// TIA Portal V20 export
FUNCTION_BLOCK "Sequence_2_TopTapeAttachment"   // FB32849, LAD
TITLE = Sequence
// Sequence template programmend in ladder logic
// stored: IsIECCheckEnabled true, MemoryReserve 100, Namespace Unit1.Em3, SetENOAutomatically true
   VAR_INPUT
      unitStatus : "LAF_typeUnitStatus";
   END_VAR
   VAR
      instSequenceLADControl { ExternalWritable := 'False'} : "LAF_ControlLadSequence";
      instSequenceLADStatus { ExternalWritable := 'False'} : "LAF_StatusLadSequence";
      statTonTime { ExternalWritable := 'False'} : Array[0..9999] of TON_TIME;
   END_VAR
   VAR_TEMP
      tempCustomerAction : Bool;   // Placeholder for possible actions
      tempDo_nothing_and_wait_for_init : Bool;   // Placeholder for doing nothing
      tempSafeStateCondition : Bool;   // Temp Condition for the equipment module to be in a safe state
   END_VAR
   VAR CONSTANT
      delayTime : Time := T#100ms;
      STEP_IDLE : DInt := 1;
      JOB_1_STEP_00 : DInt := 100;
      JOB_1_STEP_01 : DInt := 101;
      JOB_1_STEP_10 : DInt := 110;
      JOB_1_STEP_20 : DInt := 120;
      JOB_1_STEP_30 : DInt := 130;
      JOB_1_STEP_40 : DInt := 140;
      JOB_1_STEP_50 : DInt := 150;
      JOB_1_STEP_60 : DInt := 160;
      JOB_1_STEP_70 : DInt := 170;
      JOB_1_STEP_80 : DInt := 180;
      JOB_1_STEP_90 : DInt := 190;
      JOB_2_STEP_00 : DInt := 200;
      JOB_2_STEP_01 : DInt := 201;
      JOB_2_STEP_10 : DInt := 210;
      JOB_2_STEP_20 : DInt := 220;
      JOB_2_STEP_30 : DInt := 230;
      JOB_2_STEP_40 : DInt := 240;
      JOB_2_STEP_41 : DInt := 241;
      JOB_2_STEP_42 : DInt := 242;
      JOB_2_STEP_50 : DInt := 250;
      JOB_2_STEP_60 : DInt := 260;
      JOB_2_STEP_70 : DInt := 270;
      JOB_2_STEP_80 : DInt := 280;
      JOB_2_STEP_90 : DInt := 290;
      JOB_3_STEP_00 : DInt := 300;
      JOB_3_STEP_01 : DInt := 301;
      JOB_3_STEP_10 : DInt := 310;
      JOB_3_STEP_20 : DInt := 320;
      JOB_3_STEP_30 : DInt := 330;
      JOB_3_STEP_40 : DInt := 340;
      JOB_3_STEP_50 : DInt := 350;
      JOB_3_STEP_60 : DInt := 360;
      JOB_3_STEP_70 : DInt := 370;
      JOB_3_STEP_80 : DInt := 380;
      JOB_3_STEP_90 : DInt := 390;
      JOB_4_STEP_00 : DInt := 400;
      JOB_4_STEP_01 : DInt := 401;
      JOB_4_STEP_10 : DInt := 410;
      JOB_4_STEP_20 : DInt := 420;
      JOB_4_STEP_30 : DInt := 430;
      JOB_4_STEP_40 : DInt := 440;
      JOB_4_STEP_50 : DInt := 450;
      JOB_4_STEP_60 : DInt := 460;
      JOB_4_STEP_70 : DInt := 470;
      JOB_4_STEP_80 : DInt := 480;
      JOB_4_STEP_90 : DInt := 490;
      JOB_5_STEP_01 : DInt := 501;
      JOB_5_STEP_10 : DInt := 510;
      JOB_5_STEP_20 : DInt := 520;
      JOB_5_STEP_30 : DInt := 530;
      JOB_5_STEP_40 : DInt := 540;
      JOB_5_STEP_50 : DInt := 550;
      JOB_5_STEP_60 : DInt := 560;
      JOB_5_STEP_70 : DInt := 570;
      JOB_5_STEP_80 : DInt := 580;
      JOB_5_STEP_90 : DInt := 590;
      JOB_12_STEP_10 : DInt := 1210;
      JOB_12_STEP_20 : DInt := 1220;
      JOB_12_STEP_30 : DInt := 1230;
      JOB_12_STEP_40 : DInt := 1240;
      JOB_12_STEP_50 : DInt := 1250;
      JOB_12_STEP_60 : DInt := 1260;
      JOB_12_STEP_70 : DInt := 1270;
      JOB_12_STEP_80 : DInt := 1280;
      JOB_12_STEP_90 : DInt := 1290;
      JOB_13_STEP_00 : DInt := 1300;
      JOB_13_STEP_10 : DInt := 1310;
      JOB_13_STEP_20 : DInt := 1320;
      JOB_13_STEP_30 : DInt := 1330;
      JOB_13_STEP_40 : DInt := 1340;
      JOB_13_STEP_50 : DInt := 1350;
      JOB_13_STEP_60 : DInt := 1360;
      JOB_13_STEP_70 : DInt := 1370;
      JOB_13_STEP_80 : DInt := 1380;
      JOB_13_STEP_90 : DInt := 1390;
      STEP_IMMEDIATE_STOP : DInt := 9001;   // Step executed when an immediate stop command is triggered for the sequence (i.e. when unit is in state aborting)
      TO_DO_INSERT_ACTIONS_HERE : Bool := TRUE;   // Template : Add actions
      TO_DO_INSERT_CONDITION_FOR_TRANSITION_HERE : Bool := TRUE;   // Template : Add conditions
   END_VAR
   VAR_TEMP   // added for the SCL form of the ladder/FBD networks
      _w1 : Bool;
   END_VAR
BEGIN

REGION Network 1: BLOCK INFO HEADER
   // (company) / (C) Copyright (year)
   // ---------------------------------------------------------------------------------
   // Title:                             (Title of this block)
   // Comment/Function: (that is implemented in the block)
   // Library/Family:           (that the source is dedicated to)
   // Author:                        (department / person in charge / contact)
   // Target System:          (test system with FW version)
   // Engineering:              TIA Portal (SW version)
   // Restrictions:               (OB types, etc.)
   // Requirements:           (hardware, technological package, etc.)
   // ---------------------------------------------------------------------------------
   // Change log table:
   // Version          | Date             | Signature      | Expert in charge  | Changes applied ------------------------|----------------------|-------------------------|--------------------------------|-----------------------
   // 001.000.000 | yyyy-mm-dd | 0x00000000 | (name of expert) | First released version
END_REGION

REGION Network 2: DESCRIPTION
   // This is a template block provided by the Automation Framework. It can be used to create an own project.
   // The Block Info Header is prepared to put in your own data.
   // Description of the block could be added here and the docu created by Code2Docu.
END_REGION

REGION Network 3: *************** CONTROL **********************
END_REGION

REGION Network 4: Sequence Control ("Enter your Sequins number here")
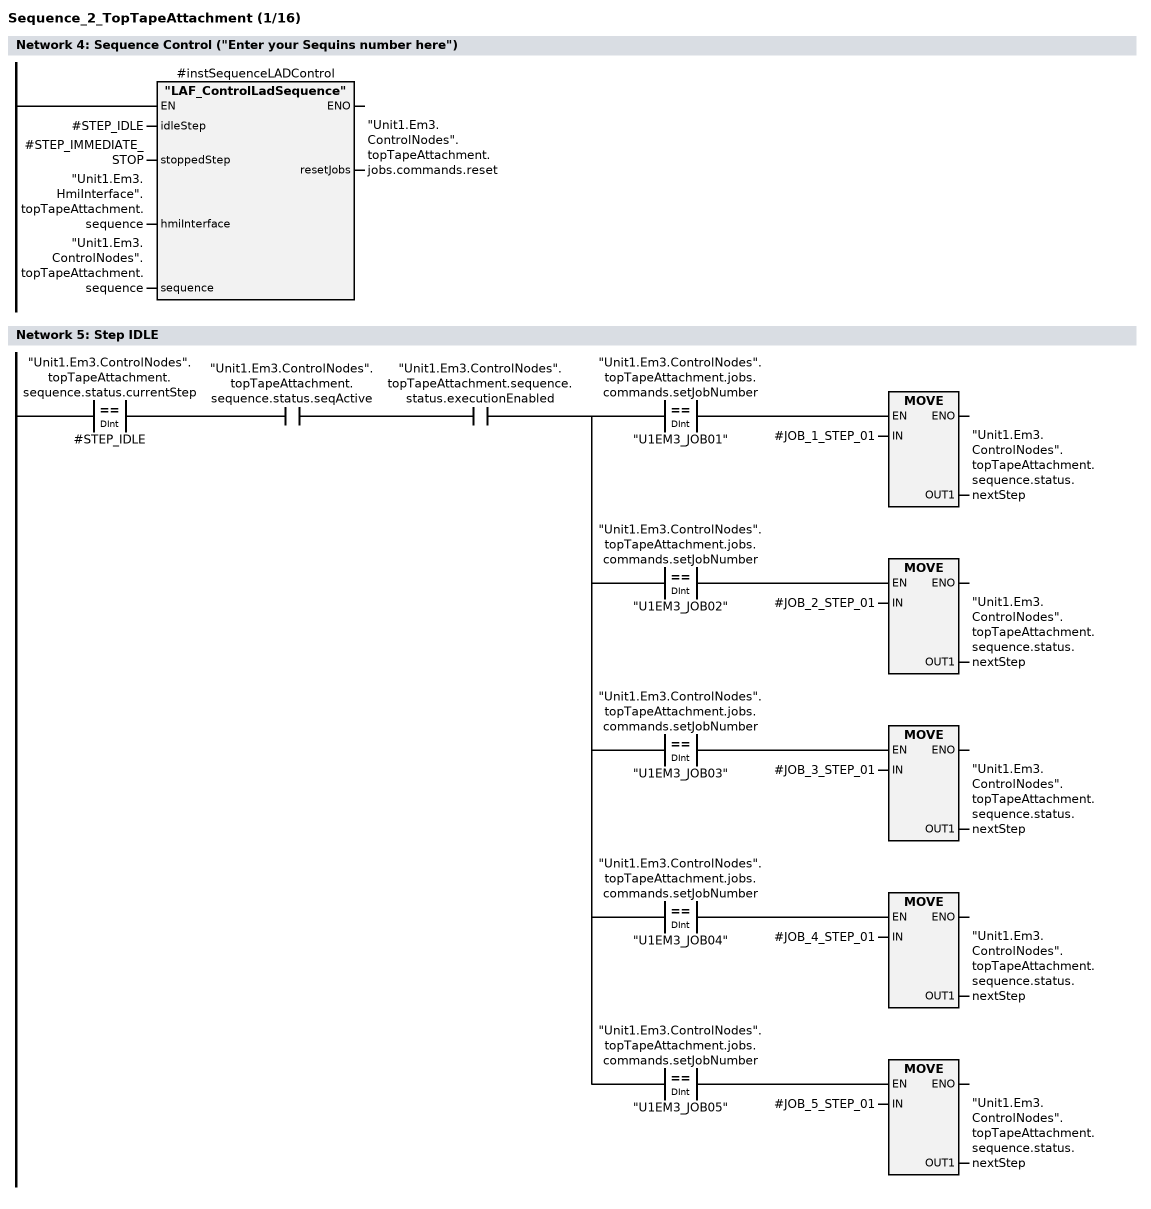
   RUNG wire#powerrail
      #instSequenceLADControl(idleStep := #STEP_IDLE, stoppedStep := #STEP_IMMEDIATE_STOP, hmiInterface := "Unit1.Em3.HmiInterface".topTapeAttachment.sequence, sequence := "Unit1.Em3.ControlNodes".topTapeAttachment.sequence, resetJobs => "Unit1.Em3.ControlNodes".topTapeAttachment.jobs.commands.reset)
   END_RUNG
   // the same network as SCL:
   #instSequenceLADControl(idleStep := #STEP_IDLE,   // "LAF_ControlLadSequence"
                           stoppedStep := #STEP_IMMEDIATE_STOP,
                           hmiInterface := "Unit1.Em3.HmiInterface".topTapeAttachment.sequence,
                           sequence := "Unit1.Em3.ControlNodes".topTapeAttachment.sequence,
                           resetJobs => "Unit1.Em3.ControlNodes".topTapeAttachment.jobs.commands.reset);
END_REGION

REGION Network 5: Step IDLE
   RUNG wire#powerrail
      { S7_Templates := "SrcType := DInt" } EQ_Contact(in1 := "Unit1.Em3.ControlNodes".topTapeAttachment.sequence.status.currentStep, in2 := #STEP_IDLE)
      Contact( "Unit1.Em3.ControlNodes".topTapeAttachment.sequence.status.seqActive )
      Contact( "Unit1.Em3.ControlNodes".topTapeAttachment.sequence.status.executionEnabled )
      wire#w1
      { S7_Templates := "SrcType := DInt" } EQ_Contact(in1 := "Unit1.Em3.ControlNodes".topTapeAttachment.jobs.commands.setJobNumber, in2 := "U1EM3_JOB01")
      Move(in := #JOB_1_STEP_01, out1 => "Unit1.Em3.ControlNodes".topTapeAttachment.sequence.status.nextStep)
   END_RUNG
   RUNG wire#w1
      { S7_Templates := "SrcType := DInt" } EQ_Contact(in1 := "Unit1.Em3.ControlNodes".topTapeAttachment.jobs.commands.setJobNumber, in2 := "U1EM3_JOB02")
      Move(in := #JOB_2_STEP_01, out1 => "Unit1.Em3.ControlNodes".topTapeAttachment.sequence.status.nextStep)
   END_RUNG
   RUNG wire#w1
      { S7_Templates := "SrcType := DInt" } EQ_Contact(in1 := "Unit1.Em3.ControlNodes".topTapeAttachment.jobs.commands.setJobNumber, in2 := "U1EM3_JOB03")
      Move(in := #JOB_3_STEP_01, out1 => "Unit1.Em3.ControlNodes".topTapeAttachment.sequence.status.nextStep)
   END_RUNG
   RUNG wire#w1
      { S7_Templates := "SrcType := DInt" } EQ_Contact(in1 := "Unit1.Em3.ControlNodes".topTapeAttachment.jobs.commands.setJobNumber, in2 := "U1EM3_JOB04")
      Move(in := #JOB_4_STEP_01, out1 => "Unit1.Em3.ControlNodes".topTapeAttachment.sequence.status.nextStep)
   END_RUNG
   RUNG wire#w1
      { S7_Templates := "SrcType := DInt" } EQ_Contact(in1 := "Unit1.Em3.ControlNodes".topTapeAttachment.jobs.commands.setJobNumber, in2 := "U1EM3_JOB05")
      Move(in := #JOB_5_STEP_01, out1 => "Unit1.Em3.ControlNodes".topTapeAttachment.sequence.status.nextStep)
   END_RUNG
   // the same network as SCL:
   #_w1 := ("Unit1.Em3.ControlNodes".topTapeAttachment.sequence.status.currentStep = #STEP_IDLE) AND "Unit1.Em3.ControlNodes".topTapeAttachment.sequence.status.seqActive AND "Unit1.Em3.ControlNodes".topTapeAttachment.sequence.status.executionEnabled;
   IF #_w1 AND ("Unit1.Em3.ControlNodes".topTapeAttachment.jobs.commands.setJobNumber = "U1EM3_JOB01") THEN
       "Unit1.Em3.ControlNodes".topTapeAttachment.sequence.status.nextStep := #JOB_1_STEP_01;
   END_IF;
   IF #_w1 AND ("Unit1.Em3.ControlNodes".topTapeAttachment.jobs.commands.setJobNumber = "U1EM3_JOB02") THEN
       "Unit1.Em3.ControlNodes".topTapeAttachment.sequence.status.nextStep := #JOB_2_STEP_01;
   END_IF;
   IF #_w1 AND ("Unit1.Em3.ControlNodes".topTapeAttachment.jobs.commands.setJobNumber = "U1EM3_JOB03") THEN
       "Unit1.Em3.ControlNodes".topTapeAttachment.sequence.status.nextStep := #JOB_3_STEP_01;
   END_IF;
   IF #_w1 AND ("Unit1.Em3.ControlNodes".topTapeAttachment.jobs.commands.setJobNumber = "U1EM3_JOB04") THEN
       "Unit1.Em3.ControlNodes".topTapeAttachment.sequence.status.nextStep := #JOB_4_STEP_01;
   END_IF;
   IF #_w1 AND ("Unit1.Em3.ControlNodes".topTapeAttachment.jobs.commands.setJobNumber = "U1EM3_JOB05") THEN
       "Unit1.Em3.ControlNodes".topTapeAttachment.sequence.status.nextStep := #JOB_5_STEP_01;
   END_IF;
END_REGION

REGION Network 6: *************** JOB[1] EM HOMING *************************
END_REGION

REGION Network 7: Step[101] : JOB[1] Condition
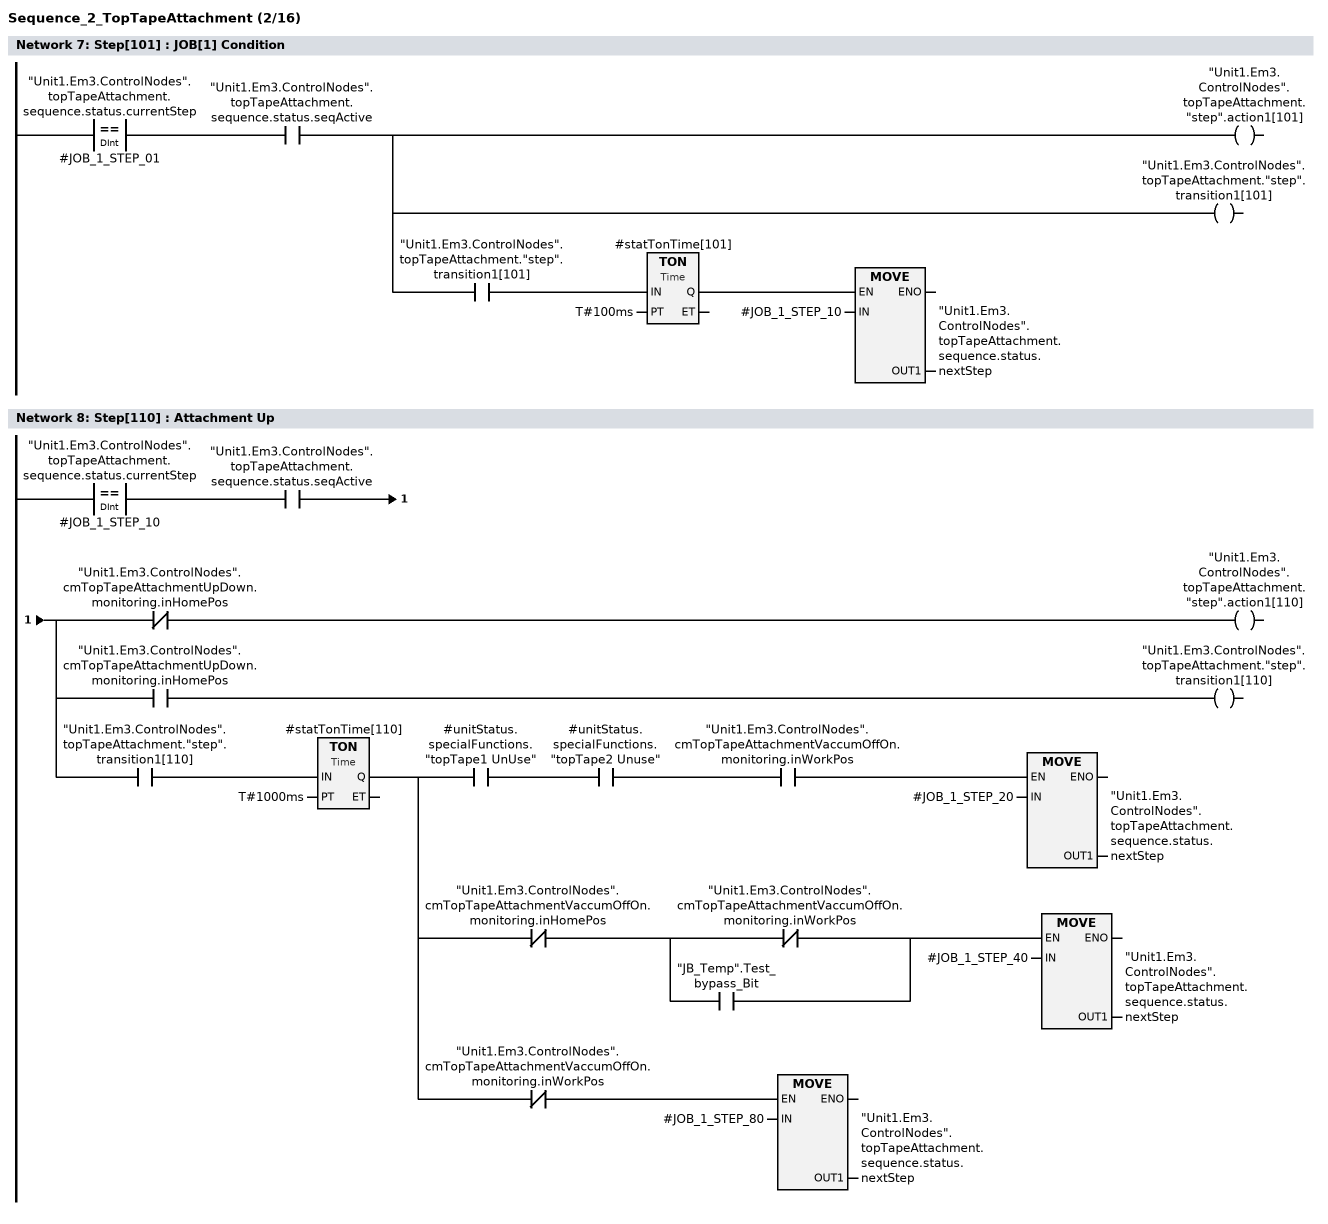
   RUNG wire#powerrail
      { S7_Templates := "SrcType := DInt" } EQ_Contact(in1 := "Unit1.Em3.ControlNodes".topTapeAttachment.sequence.status.currentStep, in2 := #JOB_1_STEP_01)
      Contact( "Unit1.Em3.ControlNodes".topTapeAttachment.sequence.status.seqActive )
      wire#w1
      Coil( "Unit1.Em3.ControlNodes".topTapeAttachment."step".action1[101] )
   END_RUNG
   RUNG wire#w1
      Coil( "Unit1.Em3.ControlNodes".topTapeAttachment."step".transition1[101] )
   END_RUNG
   RUNG wire#w1
      Contact( "Unit1.Em3.ControlNodes".topTapeAttachment."step".transition1[101] )
      { S7_Templates := "time_type := Time" } #statTonTime[101].TON(pt := T#100ms, et =>)
      Move(in := #JOB_1_STEP_10, out1 => "Unit1.Em3.ControlNodes".topTapeAttachment.sequence.status.nextStep)
   END_RUNG
   // the same network as SCL:
   "Unit1.Em3.ControlNodes".topTapeAttachment."step".action1[101] := ("Unit1.Em3.ControlNodes".topTapeAttachment.sequence.status.currentStep = #JOB_1_STEP_01) AND "Unit1.Em3.ControlNodes".topTapeAttachment.sequence.status.seqActive;
   "Unit1.Em3.ControlNodes".topTapeAttachment."step".transition1[101] := ("Unit1.Em3.ControlNodes".topTapeAttachment.sequence.status.currentStep = #JOB_1_STEP_01) AND "Unit1.Em3.ControlNodes".topTapeAttachment.sequence.status.seqActive;
   #statTonTime[101].TON(IN := ("Unit1.Em3.ControlNodes".topTapeAttachment.sequence.status.currentStep = #JOB_1_STEP_01) AND "Unit1.Em3.ControlNodes".topTapeAttachment.sequence.status.seqActive AND "Unit1.Em3.ControlNodes".topTapeAttachment."step".transition1[101],
                         PT := T#100ms);
   IF #statTonTime[101].Q THEN
       "Unit1.Em3.ControlNodes".topTapeAttachment.sequence.status.nextStep := #JOB_1_STEP_10;
   END_IF;
END_REGION

REGION Network 8: Step[110] : Attachment Up
   RUNG wire#powerrail
      { S7_Templates := "SrcType := DInt" } EQ_Contact(in1 := "Unit1.Em3.ControlNodes".topTapeAttachment.sequence.status.currentStep, in2 := #JOB_1_STEP_10)
      Contact( "Unit1.Em3.ControlNodes".topTapeAttachment.sequence.status.seqActive )
      wire#w1
      I_Contact( "Unit1.Em3.ControlNodes".cmTopTapeAttachmentUpDown.monitoring.inHomePos )
      Coil( "Unit1.Em3.ControlNodes".topTapeAttachment."step".action1[110] )
   END_RUNG
   RUNG wire#w1
      Contact( "Unit1.Em3.ControlNodes".cmTopTapeAttachmentUpDown.monitoring.inHomePos )
      Coil( "Unit1.Em3.ControlNodes".topTapeAttachment."step".transition1[110] )
   END_RUNG
   RUNG wire#w1
      Contact( "Unit1.Em3.ControlNodes".topTapeAttachment."step".transition1[110] )
      { S7_Templates := "time_type := Time" } #statTonTime[110].TON(pt := T#1000ms, et =>)
      wire#w2
      Contact( #unitStatus.specialFunctions."topTape1 UnUse" )
      Contact( #unitStatus.specialFunctions."topTape2 Unuse" )
      Contact( "Unit1.Em3.ControlNodes".cmTopTapeAttachmentVaccumOffOn.monitoring.inWorkPos )
      Move(in := #JOB_1_STEP_20, out1 => "Unit1.Em3.ControlNodes".topTapeAttachment.sequence.status.nextStep)
   END_RUNG
   RUNG wire#w2
      I_Contact( "Unit1.Em3.ControlNodes".cmTopTapeAttachmentVaccumOffOn.monitoring.inHomePos )
      wire#w3
      I_Contact( "Unit1.Em3.ControlNodes".cmTopTapeAttachmentVaccumOffOn.monitoring.inWorkPos )
      wire#w4
      Move(in := #JOB_1_STEP_40, out1 => "Unit1.Em3.ControlNodes".topTapeAttachment.sequence.status.nextStep)
   END_RUNG
   RUNG wire#w3
      Contact( "JB_Temp".Test_bypass_Bit )
   END_RUNG wire#w4
   RUNG wire#w2
      I_Contact( "Unit1.Em3.ControlNodes".cmTopTapeAttachmentVaccumOffOn.monitoring.inWorkPos )
      Move(in := #JOB_1_STEP_80, out1 => "Unit1.Em3.ControlNodes".topTapeAttachment.sequence.status.nextStep)
   END_RUNG
   // the same network as SCL:
   #_w1 := ("Unit1.Em3.ControlNodes".topTapeAttachment.sequence.status.currentStep = #JOB_1_STEP_10) AND "Unit1.Em3.ControlNodes".topTapeAttachment.sequence.status.seqActive;
   "Unit1.Em3.ControlNodes".topTapeAttachment."step".action1[110] := #_w1 AND NOT "Unit1.Em3.ControlNodes".cmTopTapeAttachmentUpDown.monitoring.inHomePos;
   "Unit1.Em3.ControlNodes".topTapeAttachment."step".transition1[110] := #_w1 AND "Unit1.Em3.ControlNodes".cmTopTapeAttachmentUpDown.monitoring.inHomePos;
   #statTonTime[110].TON(IN := #_w1 AND "Unit1.Em3.ControlNodes".topTapeAttachment."step".transition1[110],
                         PT := T#1000ms);
   IF #statTonTime[110].Q AND #unitStatus.specialFunctions."topTape1 UnUse" AND #unitStatus.specialFunctions."topTape2 Unuse" AND "Unit1.Em3.ControlNodes".cmTopTapeAttachmentVaccumOffOn.monitoring.inWorkPos THEN
       "Unit1.Em3.ControlNodes".topTapeAttachment.sequence.status.nextStep := #JOB_1_STEP_20;
   END_IF;
   IF #statTonTime[110].Q AND NOT "Unit1.Em3.ControlNodes".cmTopTapeAttachmentVaccumOffOn.monitoring.inHomePos AND (NOT "Unit1.Em3.ControlNodes".cmTopTapeAttachmentVaccumOffOn.monitoring.inWorkPos OR "JB_Temp".Test_bypass_Bit) THEN
       "Unit1.Em3.ControlNodes".topTapeAttachment.sequence.status.nextStep := #JOB_1_STEP_40;
   END_IF;
   IF #statTonTime[110].Q AND NOT "Unit1.Em3.ControlNodes".cmTopTapeAttachmentVaccumOffOn.monitoring.inWorkPos THEN
       "Unit1.Em3.ControlNodes".topTapeAttachment.sequence.status.nextStep := #JOB_1_STEP_80;
   END_IF;
END_REGION

REGION Network 9: Step[120] : Top Tape X-Axis Remains Attach Pos
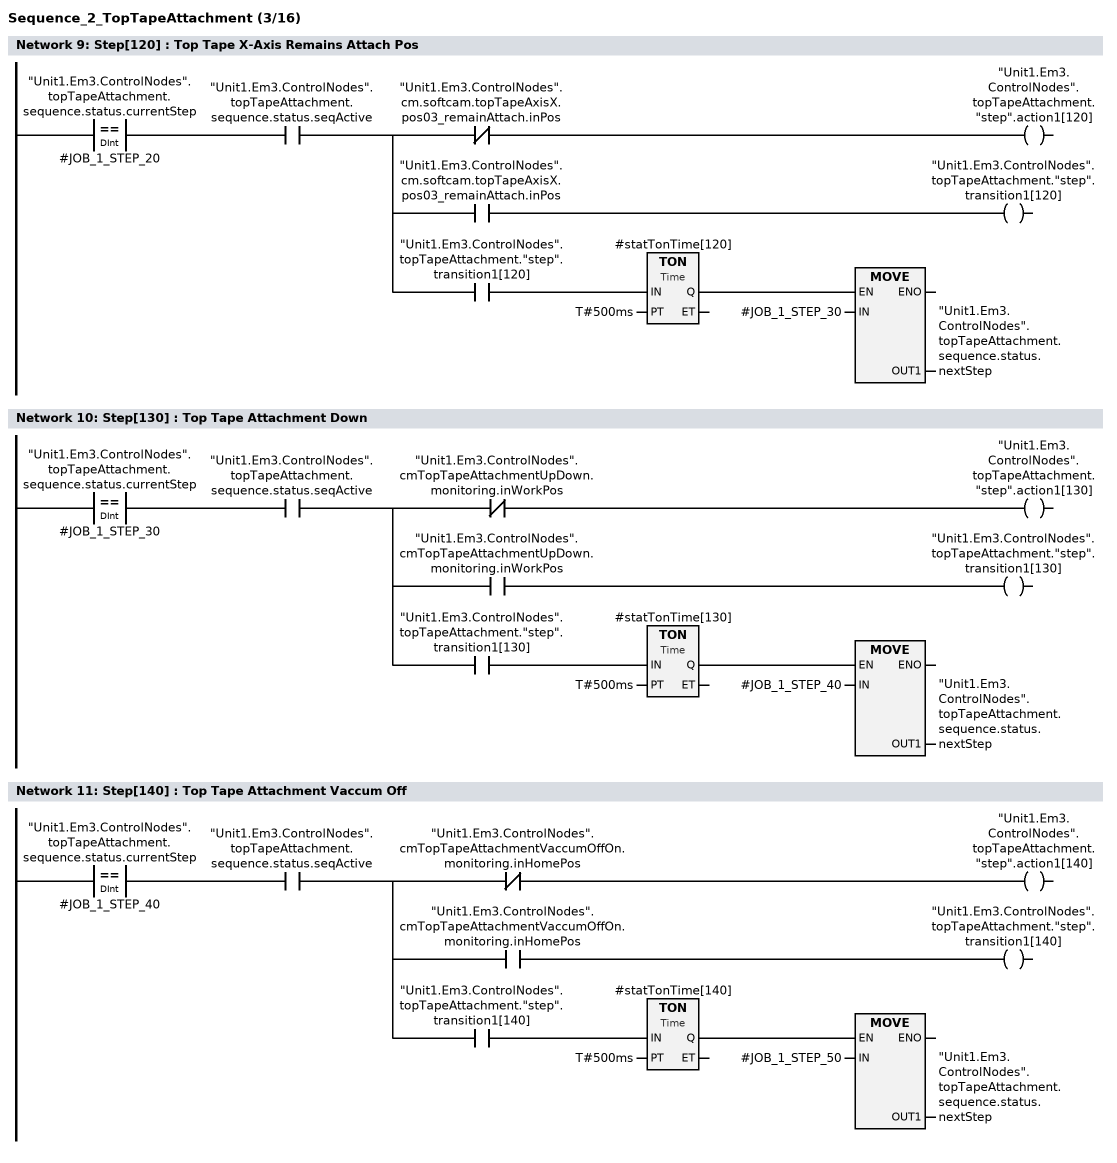
   RUNG wire#powerrail
      { S7_Templates := "SrcType := DInt" } EQ_Contact(in1 := "Unit1.Em3.ControlNodes".topTapeAttachment.sequence.status.currentStep, in2 := #JOB_1_STEP_20)
      Contact( "Unit1.Em3.ControlNodes".topTapeAttachment.sequence.status.seqActive )
      wire#w1
      I_Contact( "Unit1.Em3.ControlNodes".cm.softcam.topTapeAxisX.pos03_remainAttach.inPos )
      Coil( "Unit1.Em3.ControlNodes".topTapeAttachment."step".action1[120] )
   END_RUNG
   RUNG wire#w1
      Contact( "Unit1.Em3.ControlNodes".cm.softcam.topTapeAxisX.pos03_remainAttach.inPos )
      Coil( "Unit1.Em3.ControlNodes".topTapeAttachment."step".transition1[120] )
   END_RUNG
   RUNG wire#w1
      Contact( "Unit1.Em3.ControlNodes".topTapeAttachment."step".transition1[120] )
      { S7_Templates := "time_type := Time" } #statTonTime[120].TON(pt := T#500ms, et =>)
      Move(in := #JOB_1_STEP_30, out1 => "Unit1.Em3.ControlNodes".topTapeAttachment.sequence.status.nextStep)
   END_RUNG
   // the same network as SCL:
   #_w1 := ("Unit1.Em3.ControlNodes".topTapeAttachment.sequence.status.currentStep = #JOB_1_STEP_20) AND "Unit1.Em3.ControlNodes".topTapeAttachment.sequence.status.seqActive;
   "Unit1.Em3.ControlNodes".topTapeAttachment."step".action1[120] := #_w1 AND NOT "Unit1.Em3.ControlNodes".cm.softcam.topTapeAxisX.pos03_remainAttach.inPos;
   "Unit1.Em3.ControlNodes".topTapeAttachment."step".transition1[120] := #_w1 AND "Unit1.Em3.ControlNodes".cm.softcam.topTapeAxisX.pos03_remainAttach.inPos;
   #statTonTime[120].TON(IN := #_w1 AND "Unit1.Em3.ControlNodes".topTapeAttachment."step".transition1[120],
                         PT := T#500ms);
   IF #statTonTime[120].Q THEN
       "Unit1.Em3.ControlNodes".topTapeAttachment.sequence.status.nextStep := #JOB_1_STEP_30;
   END_IF;
END_REGION

REGION Network 10: Step[130] : Top Tape Attachment Down
   RUNG wire#powerrail
      { S7_Templates := "SrcType := DInt" } EQ_Contact(in1 := "Unit1.Em3.ControlNodes".topTapeAttachment.sequence.status.currentStep, in2 := #JOB_1_STEP_30)
      Contact( "Unit1.Em3.ControlNodes".topTapeAttachment.sequence.status.seqActive )
      wire#w1
      I_Contact( "Unit1.Em3.ControlNodes".cmTopTapeAttachmentUpDown.monitoring.inWorkPos )
      Coil( "Unit1.Em3.ControlNodes".topTapeAttachment."step".action1[130] )
   END_RUNG
   RUNG wire#w1
      Contact( "Unit1.Em3.ControlNodes".cmTopTapeAttachmentUpDown.monitoring.inWorkPos )
      Coil( "Unit1.Em3.ControlNodes".topTapeAttachment."step".transition1[130] )
   END_RUNG
   RUNG wire#w1
      Contact( "Unit1.Em3.ControlNodes".topTapeAttachment."step".transition1[130] )
      { S7_Templates := "time_type := Time" } #statTonTime[130].TON(pt := T#500ms, et =>)
      Move(in := #JOB_1_STEP_40, out1 => "Unit1.Em3.ControlNodes".topTapeAttachment.sequence.status.nextStep)
   END_RUNG
   // the same network as SCL:
   #_w1 := ("Unit1.Em3.ControlNodes".topTapeAttachment.sequence.status.currentStep = #JOB_1_STEP_30) AND "Unit1.Em3.ControlNodes".topTapeAttachment.sequence.status.seqActive;
   "Unit1.Em3.ControlNodes".topTapeAttachment."step".action1[130] := #_w1 AND NOT "Unit1.Em3.ControlNodes".cmTopTapeAttachmentUpDown.monitoring.inWorkPos;
   "Unit1.Em3.ControlNodes".topTapeAttachment."step".transition1[130] := #_w1 AND "Unit1.Em3.ControlNodes".cmTopTapeAttachmentUpDown.monitoring.inWorkPos;
   #statTonTime[130].TON(IN := #_w1 AND "Unit1.Em3.ControlNodes".topTapeAttachment."step".transition1[130],
                         PT := T#500ms);
   IF #statTonTime[130].Q THEN
       "Unit1.Em3.ControlNodes".topTapeAttachment.sequence.status.nextStep := #JOB_1_STEP_40;
   END_IF;
END_REGION

REGION Network 11: Step[140] : Top Tape Attachment Vaccum Off
   RUNG wire#powerrail
      { S7_Templates := "SrcType := DInt" } EQ_Contact(in1 := "Unit1.Em3.ControlNodes".topTapeAttachment.sequence.status.currentStep, in2 := #JOB_1_STEP_40)
      Contact( "Unit1.Em3.ControlNodes".topTapeAttachment.sequence.status.seqActive )
      wire#w1
      I_Contact( "Unit1.Em3.ControlNodes".cmTopTapeAttachmentVaccumOffOn.monitoring.inHomePos )
      Coil( "Unit1.Em3.ControlNodes".topTapeAttachment."step".action1[140] )
   END_RUNG
   RUNG wire#w1
      Contact( "Unit1.Em3.ControlNodes".cmTopTapeAttachmentVaccumOffOn.monitoring.inHomePos )
      Coil( "Unit1.Em3.ControlNodes".topTapeAttachment."step".transition1[140] )
   END_RUNG
   RUNG wire#w1
      Contact( "Unit1.Em3.ControlNodes".topTapeAttachment."step".transition1[140] )
      { S7_Templates := "time_type := Time" } #statTonTime[140].TON(pt := T#500ms, et =>)
      Move(in := #JOB_1_STEP_50, out1 => "Unit1.Em3.ControlNodes".topTapeAttachment.sequence.status.nextStep)
   END_RUNG
   // the same network as SCL:
   #_w1 := ("Unit1.Em3.ControlNodes".topTapeAttachment.sequence.status.currentStep = #JOB_1_STEP_40) AND "Unit1.Em3.ControlNodes".topTapeAttachment.sequence.status.seqActive;
   "Unit1.Em3.ControlNodes".topTapeAttachment."step".action1[140] := #_w1 AND NOT "Unit1.Em3.ControlNodes".cmTopTapeAttachmentVaccumOffOn.monitoring.inHomePos;
   "Unit1.Em3.ControlNodes".topTapeAttachment."step".transition1[140] := #_w1 AND "Unit1.Em3.ControlNodes".cmTopTapeAttachmentVaccumOffOn.monitoring.inHomePos;
   #statTonTime[140].TON(IN := #_w1 AND "Unit1.Em3.ControlNodes".topTapeAttachment."step".transition1[140],
                         PT := T#500ms);
   IF #statTonTime[140].Q THEN
       "Unit1.Em3.ControlNodes".topTapeAttachment.sequence.status.nextStep := #JOB_1_STEP_50;
   END_IF;
END_REGION

REGION Network 12: Step[150] : Top Tape Attachment Up
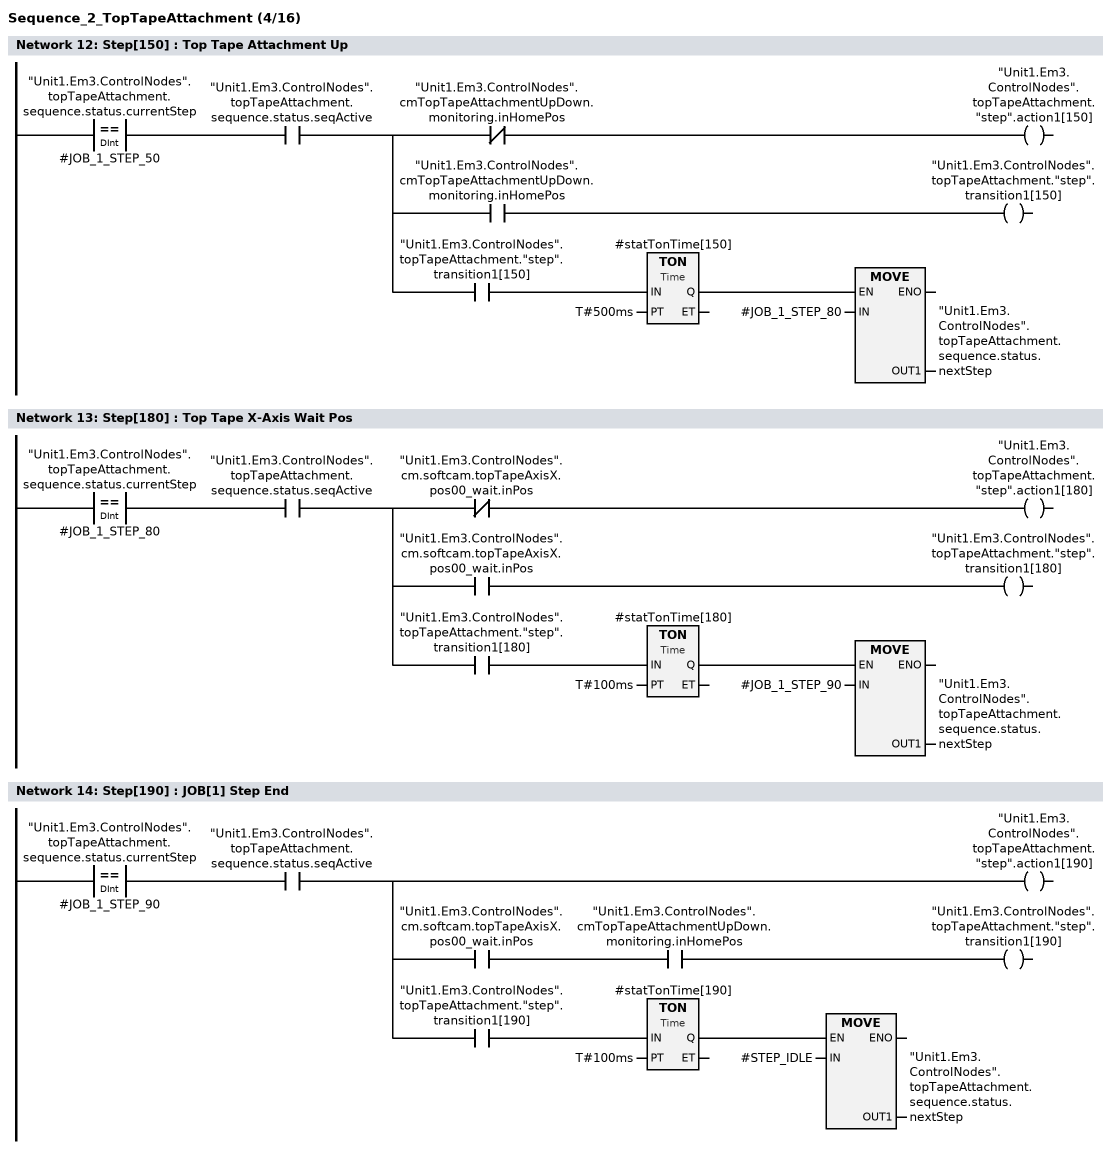
   RUNG wire#powerrail
      { S7_Templates := "SrcType := DInt" } EQ_Contact(in1 := "Unit1.Em3.ControlNodes".topTapeAttachment.sequence.status.currentStep, in2 := #JOB_1_STEP_50)
      Contact( "Unit1.Em3.ControlNodes".topTapeAttachment.sequence.status.seqActive )
      wire#w1
      I_Contact( "Unit1.Em3.ControlNodes".cmTopTapeAttachmentUpDown.monitoring.inHomePos )
      Coil( "Unit1.Em3.ControlNodes".topTapeAttachment."step".action1[150] )
   END_RUNG
   RUNG wire#w1
      Contact( "Unit1.Em3.ControlNodes".cmTopTapeAttachmentUpDown.monitoring.inHomePos )
      Coil( "Unit1.Em3.ControlNodes".topTapeAttachment."step".transition1[150] )
   END_RUNG
   RUNG wire#w1
      Contact( "Unit1.Em3.ControlNodes".topTapeAttachment."step".transition1[150] )
      { S7_Templates := "time_type := Time" } #statTonTime[150].TON(pt := T#500ms, et =>)
      Move(in := #JOB_1_STEP_80, out1 => "Unit1.Em3.ControlNodes".topTapeAttachment.sequence.status.nextStep)
   END_RUNG
   // the same network as SCL:
   #_w1 := ("Unit1.Em3.ControlNodes".topTapeAttachment.sequence.status.currentStep = #JOB_1_STEP_50) AND "Unit1.Em3.ControlNodes".topTapeAttachment.sequence.status.seqActive;
   "Unit1.Em3.ControlNodes".topTapeAttachment."step".action1[150] := #_w1 AND NOT "Unit1.Em3.ControlNodes".cmTopTapeAttachmentUpDown.monitoring.inHomePos;
   "Unit1.Em3.ControlNodes".topTapeAttachment."step".transition1[150] := #_w1 AND "Unit1.Em3.ControlNodes".cmTopTapeAttachmentUpDown.monitoring.inHomePos;
   #statTonTime[150].TON(IN := #_w1 AND "Unit1.Em3.ControlNodes".topTapeAttachment."step".transition1[150],
                         PT := T#500ms);
   IF #statTonTime[150].Q THEN
       "Unit1.Em3.ControlNodes".topTapeAttachment.sequence.status.nextStep := #JOB_1_STEP_80;
   END_IF;
END_REGION

REGION Network 13: Step[180] : Top Tape X-Axis Wait Pos
   RUNG wire#powerrail
      { S7_Templates := "SrcType := DInt" } EQ_Contact(in1 := "Unit1.Em3.ControlNodes".topTapeAttachment.sequence.status.currentStep, in2 := #JOB_1_STEP_80)
      Contact( "Unit1.Em3.ControlNodes".topTapeAttachment.sequence.status.seqActive )
      wire#w1
      I_Contact( "Unit1.Em3.ControlNodes".cm.softcam.topTapeAxisX.pos00_wait.inPos )
      Coil( "Unit1.Em3.ControlNodes".topTapeAttachment."step".action1[180] )
   END_RUNG
   RUNG wire#w1
      Contact( "Unit1.Em3.ControlNodes".cm.softcam.topTapeAxisX.pos00_wait.inPos )
      Coil( "Unit1.Em3.ControlNodes".topTapeAttachment."step".transition1[180] )
   END_RUNG
   RUNG wire#w1
      Contact( "Unit1.Em3.ControlNodes".topTapeAttachment."step".transition1[180] )
      { S7_Templates := "time_type := Time" } #statTonTime[180].TON(pt := T#100ms, et =>)
      Move(in := #JOB_1_STEP_90, out1 => "Unit1.Em3.ControlNodes".topTapeAttachment.sequence.status.nextStep)
   END_RUNG
   // the same network as SCL:
   #_w1 := ("Unit1.Em3.ControlNodes".topTapeAttachment.sequence.status.currentStep = #JOB_1_STEP_80) AND "Unit1.Em3.ControlNodes".topTapeAttachment.sequence.status.seqActive;
   "Unit1.Em3.ControlNodes".topTapeAttachment."step".action1[180] := #_w1 AND NOT "Unit1.Em3.ControlNodes".cm.softcam.topTapeAxisX.pos00_wait.inPos;
   "Unit1.Em3.ControlNodes".topTapeAttachment."step".transition1[180] := #_w1 AND "Unit1.Em3.ControlNodes".cm.softcam.topTapeAxisX.pos00_wait.inPos;
   #statTonTime[180].TON(IN := #_w1 AND "Unit1.Em3.ControlNodes".topTapeAttachment."step".transition1[180],
                         PT := T#100ms);
   IF #statTonTime[180].Q THEN
       "Unit1.Em3.ControlNodes".topTapeAttachment.sequence.status.nextStep := #JOB_1_STEP_90;
   END_IF;
END_REGION

REGION Network 14: Step[190] : JOB[1] Step End
   RUNG wire#powerrail
      { S7_Templates := "SrcType := DInt" } EQ_Contact(in1 := "Unit1.Em3.ControlNodes".topTapeAttachment.sequence.status.currentStep, in2 := #JOB_1_STEP_90)
      Contact( "Unit1.Em3.ControlNodes".topTapeAttachment.sequence.status.seqActive )
      wire#w1
      Coil( "Unit1.Em3.ControlNodes".topTapeAttachment."step".action1[190] )
   END_RUNG
   RUNG wire#w1
      Contact( "Unit1.Em3.ControlNodes".cm.softcam.topTapeAxisX.pos00_wait.inPos )
      Contact( "Unit1.Em3.ControlNodes".cmTopTapeAttachmentUpDown.monitoring.inHomePos )
      Coil( "Unit1.Em3.ControlNodes".topTapeAttachment."step".transition1[190] )
   END_RUNG
   RUNG wire#w1
      Contact( "Unit1.Em3.ControlNodes".topTapeAttachment."step".transition1[190] )
      { S7_Templates := "time_type := Time" } #statTonTime[190].TON(pt := T#100ms, et =>)
      Move(in := #STEP_IDLE, out1 => "Unit1.Em3.ControlNodes".topTapeAttachment.sequence.status.nextStep)
   END_RUNG
   // the same network as SCL:
   "Unit1.Em3.ControlNodes".topTapeAttachment."step".action1[190] := ("Unit1.Em3.ControlNodes".topTapeAttachment.sequence.status.currentStep = #JOB_1_STEP_90) AND "Unit1.Em3.ControlNodes".topTapeAttachment.sequence.status.seqActive;
   "Unit1.Em3.ControlNodes".topTapeAttachment."step".transition1[190] := ("Unit1.Em3.ControlNodes".topTapeAttachment.sequence.status.currentStep = #JOB_1_STEP_90) AND "Unit1.Em3.ControlNodes".topTapeAttachment.sequence.status.seqActive AND "Unit1.Em3.ControlNodes".cm.softcam.topTapeAxisX.pos00_wait.inPos AND "Unit1.Em3.ControlNodes".cmTopTapeAttachmentUpDown.monitoring.inHomePos;
   #statTonTime[190].TON(IN := ("Unit1.Em3.ControlNodes".topTapeAttachment.sequence.status.currentStep = #JOB_1_STEP_90) AND "Unit1.Em3.ControlNodes".topTapeAttachment.sequence.status.seqActive AND "Unit1.Em3.ControlNodes".topTapeAttachment."step".transition1[190],
                         PT := T#100ms);
   IF #statTonTime[190].Q THEN
       "Unit1.Em3.ControlNodes".topTapeAttachment.sequence.status.nextStep := #STEP_IDLE;
   END_IF;
END_REGION

REGION Network 15: *************** JOB[2] TOP TAPE GET=AUTO *************************
END_REGION

REGION Network 16: Step[201] : JOB[2] Condition
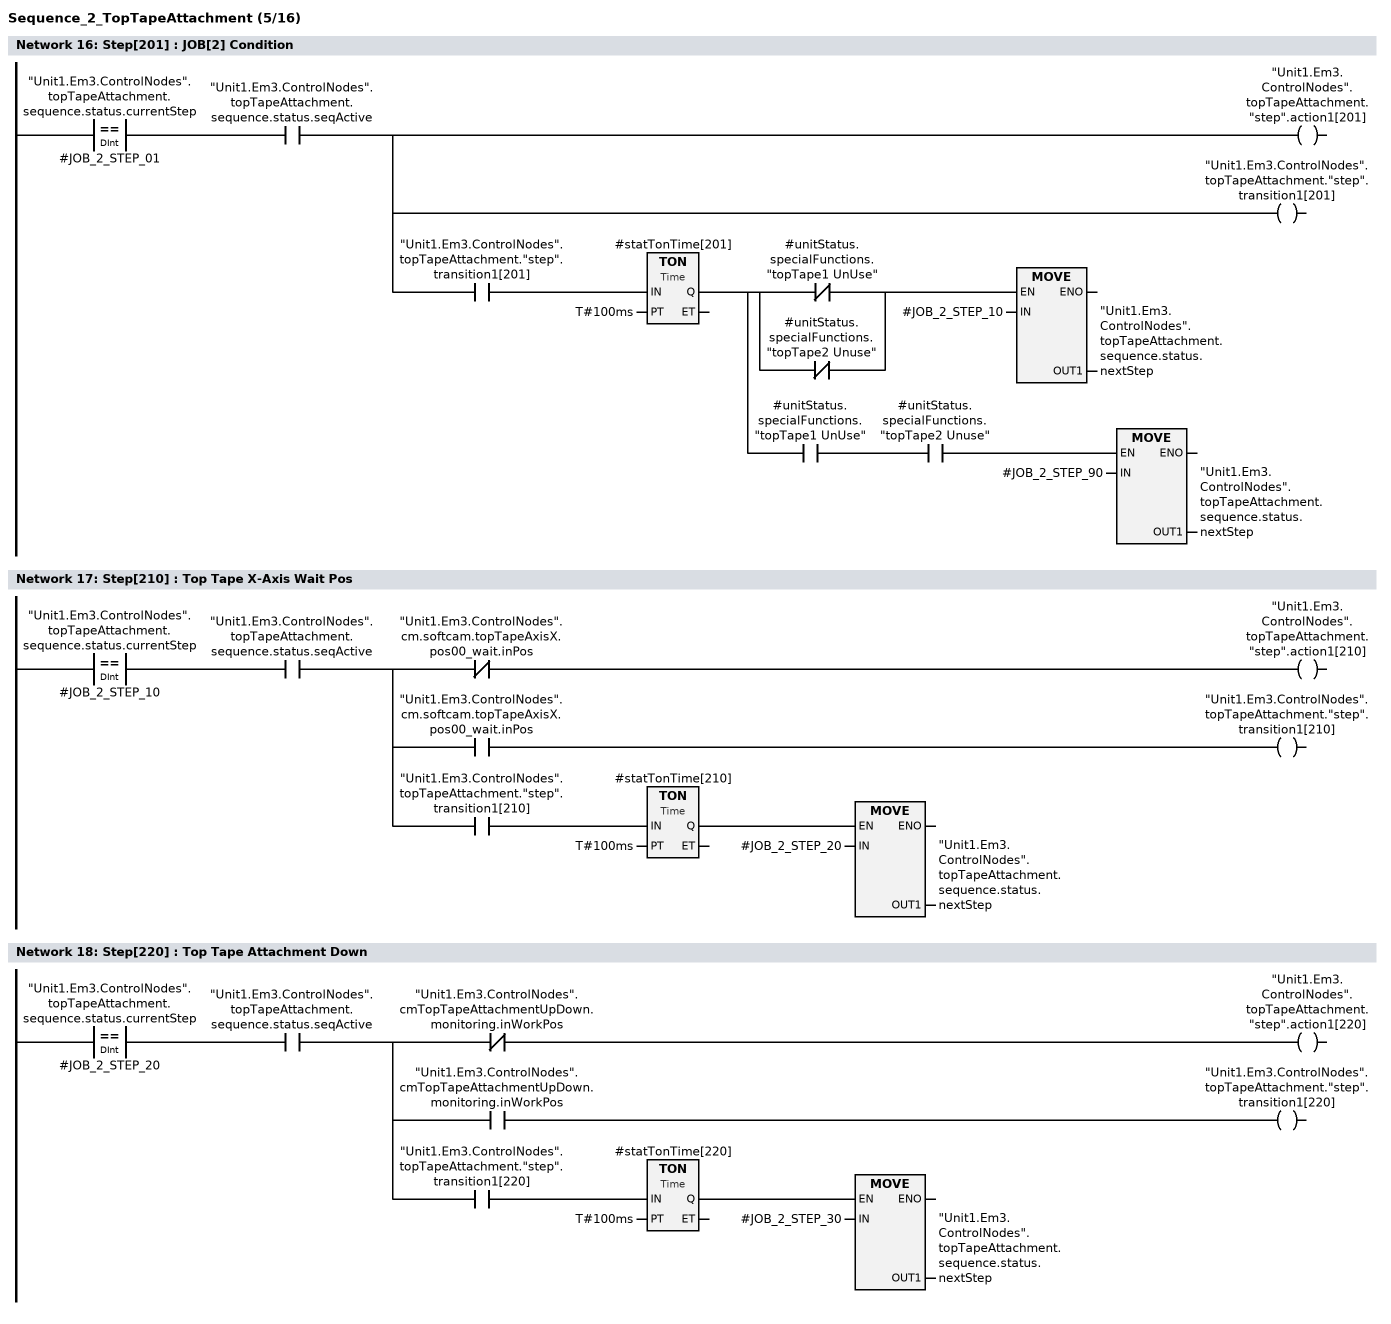
   RUNG wire#powerrail
      { S7_Templates := "SrcType := DInt" } EQ_Contact(in1 := "Unit1.Em3.ControlNodes".topTapeAttachment.sequence.status.currentStep, in2 := #JOB_2_STEP_01)
      Contact( "Unit1.Em3.ControlNodes".topTapeAttachment.sequence.status.seqActive )
      wire#w1
      Coil( "Unit1.Em3.ControlNodes".topTapeAttachment."step".action1[201] )
   END_RUNG
   RUNG wire#w1
      Coil( "Unit1.Em3.ControlNodes".topTapeAttachment."step".transition1[201] )
   END_RUNG
   RUNG wire#w1
      Contact( "Unit1.Em3.ControlNodes".topTapeAttachment."step".transition1[201] )
      { S7_Templates := "time_type := Time" } #statTonTime[201].TON(pt := T#100ms, et =>)
      wire#w2
      I_Contact( #unitStatus.specialFunctions."topTape1 UnUse" )
      wire#w3
      Move(in := #JOB_2_STEP_10, out1 => "Unit1.Em3.ControlNodes".topTapeAttachment.sequence.status.nextStep)
   END_RUNG
   RUNG wire#w2
      I_Contact( #unitStatus.specialFunctions."topTape2 Unuse" )
   END_RUNG wire#w3
   RUNG wire#w2
      Contact( #unitStatus.specialFunctions."topTape1 UnUse" )
      Contact( #unitStatus.specialFunctions."topTape2 Unuse" )
      Move(in := #JOB_2_STEP_90, out1 => "Unit1.Em3.ControlNodes".topTapeAttachment.sequence.status.nextStep)
   END_RUNG
   // the same network as SCL:
   "Unit1.Em3.ControlNodes".topTapeAttachment."step".action1[201] := ("Unit1.Em3.ControlNodes".topTapeAttachment.sequence.status.currentStep = #JOB_2_STEP_01) AND "Unit1.Em3.ControlNodes".topTapeAttachment.sequence.status.seqActive;
   "Unit1.Em3.ControlNodes".topTapeAttachment."step".transition1[201] := ("Unit1.Em3.ControlNodes".topTapeAttachment.sequence.status.currentStep = #JOB_2_STEP_01) AND "Unit1.Em3.ControlNodes".topTapeAttachment.sequence.status.seqActive;
   #statTonTime[201].TON(IN := ("Unit1.Em3.ControlNodes".topTapeAttachment.sequence.status.currentStep = #JOB_2_STEP_01) AND "Unit1.Em3.ControlNodes".topTapeAttachment.sequence.status.seqActive AND "Unit1.Em3.ControlNodes".topTapeAttachment."step".transition1[201],
                         PT := T#100ms);
   IF #statTonTime[201].Q AND (NOT #unitStatus.specialFunctions."topTape1 UnUse" OR NOT #unitStatus.specialFunctions."topTape2 Unuse") THEN
       "Unit1.Em3.ControlNodes".topTapeAttachment.sequence.status.nextStep := #JOB_2_STEP_10;
   END_IF;
   IF #statTonTime[201].Q AND #unitStatus.specialFunctions."topTape1 UnUse" AND #unitStatus.specialFunctions."topTape2 Unuse" THEN
       "Unit1.Em3.ControlNodes".topTapeAttachment.sequence.status.nextStep := #JOB_2_STEP_90;
   END_IF;
END_REGION

REGION Network 17: Step[210] : Top Tape X-Axis Wait Pos
   RUNG wire#powerrail
      { S7_Templates := "SrcType := DInt" } EQ_Contact(in1 := "Unit1.Em3.ControlNodes".topTapeAttachment.sequence.status.currentStep, in2 := #JOB_2_STEP_10)
      Contact( "Unit1.Em3.ControlNodes".topTapeAttachment.sequence.status.seqActive )
      wire#w1
      I_Contact( "Unit1.Em3.ControlNodes".cm.softcam.topTapeAxisX.pos00_wait.inPos )
      Coil( "Unit1.Em3.ControlNodes".topTapeAttachment."step".action1[210] )
   END_RUNG
   RUNG wire#w1
      Contact( "Unit1.Em3.ControlNodes".cm.softcam.topTapeAxisX.pos00_wait.inPos )
      Coil( "Unit1.Em3.ControlNodes".topTapeAttachment."step".transition1[210] )
   END_RUNG
   RUNG wire#w1
      Contact( "Unit1.Em3.ControlNodes".topTapeAttachment."step".transition1[210] )
      { S7_Templates := "time_type := Time" } #statTonTime[210].TON(pt := T#100ms, et =>)
      Move(in := #JOB_2_STEP_20, out1 => "Unit1.Em3.ControlNodes".topTapeAttachment.sequence.status.nextStep)
   END_RUNG
   // the same network as SCL:
   #_w1 := ("Unit1.Em3.ControlNodes".topTapeAttachment.sequence.status.currentStep = #JOB_2_STEP_10) AND "Unit1.Em3.ControlNodes".topTapeAttachment.sequence.status.seqActive;
   "Unit1.Em3.ControlNodes".topTapeAttachment."step".action1[210] := #_w1 AND NOT "Unit1.Em3.ControlNodes".cm.softcam.topTapeAxisX.pos00_wait.inPos;
   "Unit1.Em3.ControlNodes".topTapeAttachment."step".transition1[210] := #_w1 AND "Unit1.Em3.ControlNodes".cm.softcam.topTapeAxisX.pos00_wait.inPos;
   #statTonTime[210].TON(IN := #_w1 AND "Unit1.Em3.ControlNodes".topTapeAttachment."step".transition1[210],
                         PT := T#100ms);
   IF #statTonTime[210].Q THEN
       "Unit1.Em3.ControlNodes".topTapeAttachment.sequence.status.nextStep := #JOB_2_STEP_20;
   END_IF;
END_REGION

REGION Network 18: Step[220] : Top Tape Attachment Down
   RUNG wire#powerrail
      { S7_Templates := "SrcType := DInt" } EQ_Contact(in1 := "Unit1.Em3.ControlNodes".topTapeAttachment.sequence.status.currentStep, in2 := #JOB_2_STEP_20)
      Contact( "Unit1.Em3.ControlNodes".topTapeAttachment.sequence.status.seqActive )
      wire#w1
      I_Contact( "Unit1.Em3.ControlNodes".cmTopTapeAttachmentUpDown.monitoring.inWorkPos )
      Coil( "Unit1.Em3.ControlNodes".topTapeAttachment."step".action1[220] )
   END_RUNG
   RUNG wire#w1
      Contact( "Unit1.Em3.ControlNodes".cmTopTapeAttachmentUpDown.monitoring.inWorkPos )
      Coil( "Unit1.Em3.ControlNodes".topTapeAttachment."step".transition1[220] )
   END_RUNG
   RUNG wire#w1
      Contact( "Unit1.Em3.ControlNodes".topTapeAttachment."step".transition1[220] )
      { S7_Templates := "time_type := Time" } #statTonTime[220].TON(pt := T#100ms, et =>)
      Move(in := #JOB_2_STEP_30, out1 => "Unit1.Em3.ControlNodes".topTapeAttachment.sequence.status.nextStep)
   END_RUNG
   // the same network as SCL:
   #_w1 := ("Unit1.Em3.ControlNodes".topTapeAttachment.sequence.status.currentStep = #JOB_2_STEP_20) AND "Unit1.Em3.ControlNodes".topTapeAttachment.sequence.status.seqActive;
   "Unit1.Em3.ControlNodes".topTapeAttachment."step".action1[220] := #_w1 AND NOT "Unit1.Em3.ControlNodes".cmTopTapeAttachmentUpDown.monitoring.inWorkPos;
   "Unit1.Em3.ControlNodes".topTapeAttachment."step".transition1[220] := #_w1 AND "Unit1.Em3.ControlNodes".cmTopTapeAttachmentUpDown.monitoring.inWorkPos;
   #statTonTime[220].TON(IN := #_w1 AND "Unit1.Em3.ControlNodes".topTapeAttachment."step".transition1[220],
                         PT := T#100ms);
   IF #statTonTime[220].Q THEN
       "Unit1.Em3.ControlNodes".topTapeAttachment.sequence.status.nextStep := #JOB_2_STEP_30;
   END_IF;
END_REGION

REGION Network 19: Step[230] : Top Tape Attachment Vacuum On
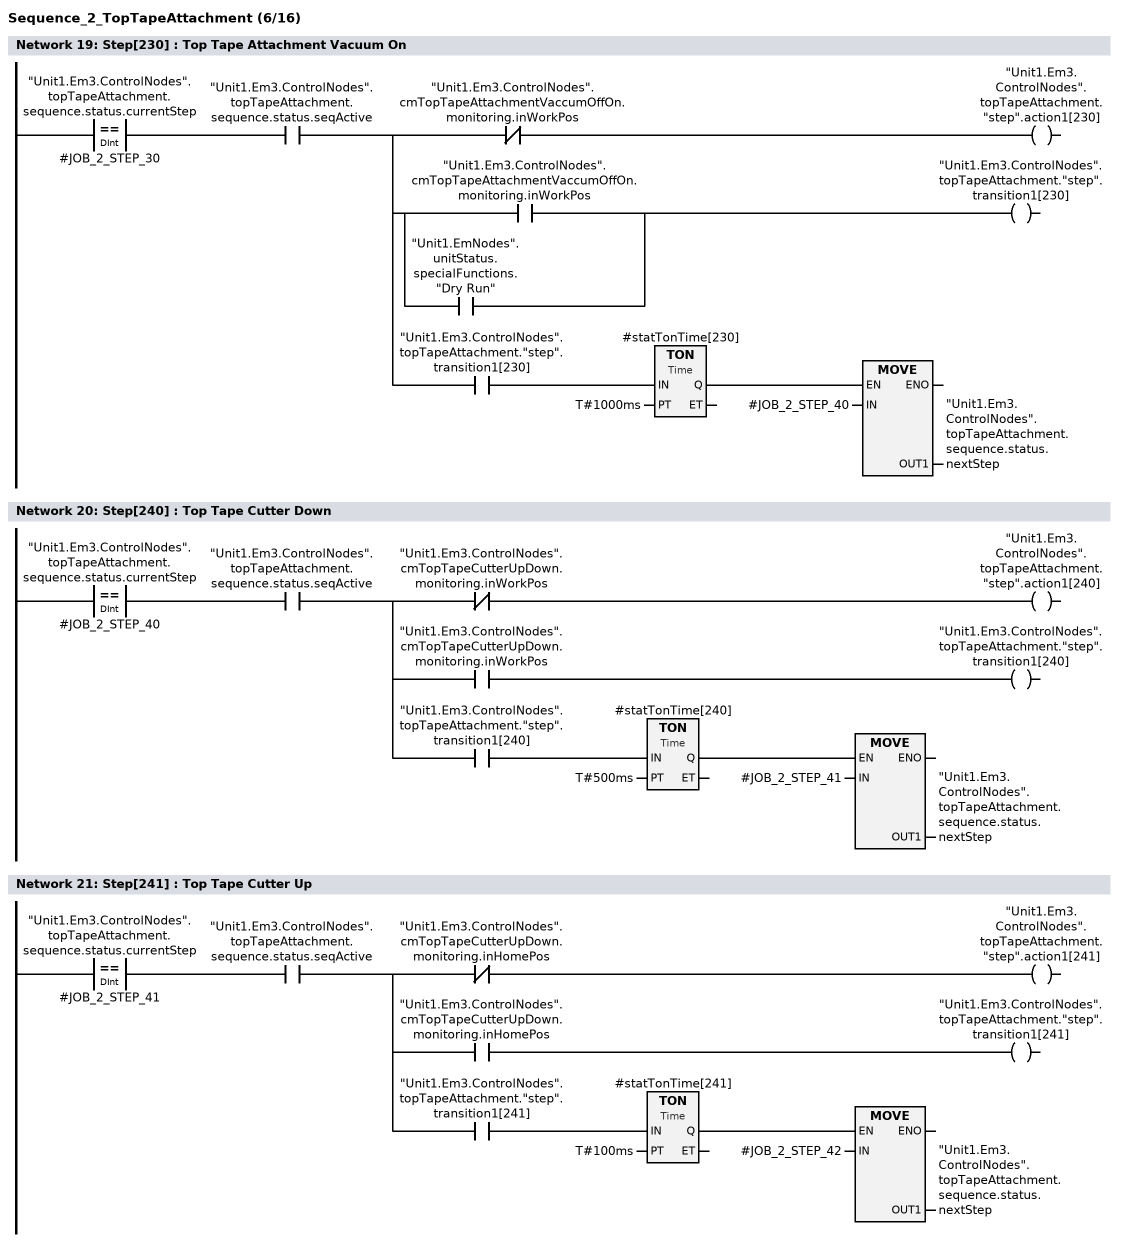
   RUNG wire#powerrail
      { S7_Templates := "SrcType := DInt" } EQ_Contact(in1 := "Unit1.Em3.ControlNodes".topTapeAttachment.sequence.status.currentStep, in2 := #JOB_2_STEP_30)
      Contact( "Unit1.Em3.ControlNodes".topTapeAttachment.sequence.status.seqActive )
      wire#w1
      I_Contact( "Unit1.Em3.ControlNodes".cmTopTapeAttachmentVaccumOffOn.monitoring.inWorkPos )
      Coil( "Unit1.Em3.ControlNodes".topTapeAttachment."step".action1[230] )
   END_RUNG
   RUNG wire#w1
      Contact( "Unit1.Em3.ControlNodes".cmTopTapeAttachmentVaccumOffOn.monitoring.inWorkPos )
      wire#w2
      Coil( "Unit1.Em3.ControlNodes".topTapeAttachment."step".transition1[230] )
   END_RUNG
   RUNG wire#w1
      Contact( "Unit1.EmNodes".unitStatus.specialFunctions."Dry Run" )
   END_RUNG wire#w2
   RUNG wire#w1
      Contact( "Unit1.Em3.ControlNodes".topTapeAttachment."step".transition1[230] )
      { S7_Templates := "time_type := Time" } #statTonTime[230].TON(pt := T#1000ms, et =>)
      Move(in := #JOB_2_STEP_40, out1 => "Unit1.Em3.ControlNodes".topTapeAttachment.sequence.status.nextStep)
   END_RUNG
   // the same network as SCL:
   #_w1 := ("Unit1.Em3.ControlNodes".topTapeAttachment.sequence.status.currentStep = #JOB_2_STEP_30) AND "Unit1.Em3.ControlNodes".topTapeAttachment.sequence.status.seqActive;
   "Unit1.Em3.ControlNodes".topTapeAttachment."step".action1[230] := #_w1 AND NOT "Unit1.Em3.ControlNodes".cmTopTapeAttachmentVaccumOffOn.monitoring.inWorkPos;
   "Unit1.Em3.ControlNodes".topTapeAttachment."step".transition1[230] := #_w1 AND ("Unit1.Em3.ControlNodes".cmTopTapeAttachmentVaccumOffOn.monitoring.inWorkPos OR "Unit1.EmNodes".unitStatus.specialFunctions."Dry Run");
   #statTonTime[230].TON(IN := #_w1 AND "Unit1.Em3.ControlNodes".topTapeAttachment."step".transition1[230],
                         PT := T#1000ms);
   IF #statTonTime[230].Q THEN
       "Unit1.Em3.ControlNodes".topTapeAttachment.sequence.status.nextStep := #JOB_2_STEP_40;
   END_IF;
END_REGION

REGION Network 20: Step[240] : Top Tape Cutter Down
   RUNG wire#powerrail
      { S7_Templates := "SrcType := DInt" } EQ_Contact(in1 := "Unit1.Em3.ControlNodes".topTapeAttachment.sequence.status.currentStep, in2 := #JOB_2_STEP_40)
      Contact( "Unit1.Em3.ControlNodes".topTapeAttachment.sequence.status.seqActive )
      wire#w1
      I_Contact( "Unit1.Em3.ControlNodes".cmTopTapeCutterUpDown.monitoring.inWorkPos )
      Coil( "Unit1.Em3.ControlNodes".topTapeAttachment."step".action1[240] )
   END_RUNG
   RUNG wire#w1
      Contact( "Unit1.Em3.ControlNodes".cmTopTapeCutterUpDown.monitoring.inWorkPos )
      Coil( "Unit1.Em3.ControlNodes".topTapeAttachment."step".transition1[240] )
   END_RUNG
   RUNG wire#w1
      Contact( "Unit1.Em3.ControlNodes".topTapeAttachment."step".transition1[240] )
      { S7_Templates := "time_type := Time" } #statTonTime[240].TON(pt := T#500ms, et =>)
      Move(in := #JOB_2_STEP_41, out1 => "Unit1.Em3.ControlNodes".topTapeAttachment.sequence.status.nextStep)
   END_RUNG
   // the same network as SCL:
   #_w1 := ("Unit1.Em3.ControlNodes".topTapeAttachment.sequence.status.currentStep = #JOB_2_STEP_40) AND "Unit1.Em3.ControlNodes".topTapeAttachment.sequence.status.seqActive;
   "Unit1.Em3.ControlNodes".topTapeAttachment."step".action1[240] := #_w1 AND NOT "Unit1.Em3.ControlNodes".cmTopTapeCutterUpDown.monitoring.inWorkPos;
   "Unit1.Em3.ControlNodes".topTapeAttachment."step".transition1[240] := #_w1 AND "Unit1.Em3.ControlNodes".cmTopTapeCutterUpDown.monitoring.inWorkPos;
   #statTonTime[240].TON(IN := #_w1 AND "Unit1.Em3.ControlNodes".topTapeAttachment."step".transition1[240],
                         PT := T#500ms);
   IF #statTonTime[240].Q THEN
       "Unit1.Em3.ControlNodes".topTapeAttachment.sequence.status.nextStep := #JOB_2_STEP_41;
   END_IF;
END_REGION

REGION Network 21: Step[241] : Top Tape Cutter Up
   RUNG wire#powerrail
      { S7_Templates := "SrcType := DInt" } EQ_Contact(in1 := "Unit1.Em3.ControlNodes".topTapeAttachment.sequence.status.currentStep, in2 := #JOB_2_STEP_41)
      Contact( "Unit1.Em3.ControlNodes".topTapeAttachment.sequence.status.seqActive )
      wire#w1
      I_Contact( "Unit1.Em3.ControlNodes".cmTopTapeCutterUpDown.monitoring.inHomePos )
      Coil( "Unit1.Em3.ControlNodes".topTapeAttachment."step".action1[241] )
   END_RUNG
   RUNG wire#w1
      Contact( "Unit1.Em3.ControlNodes".cmTopTapeCutterUpDown.monitoring.inHomePos )
      Coil( "Unit1.Em3.ControlNodes".topTapeAttachment."step".transition1[241] )
   END_RUNG
   RUNG wire#w1
      Contact( "Unit1.Em3.ControlNodes".topTapeAttachment."step".transition1[241] )
      { S7_Templates := "time_type := Time" } #statTonTime[241].TON(pt := T#100ms, et =>)
      Move(in := #JOB_2_STEP_42, out1 => "Unit1.Em3.ControlNodes".topTapeAttachment.sequence.status.nextStep)
   END_RUNG
   // the same network as SCL:
   #_w1 := ("Unit1.Em3.ControlNodes".topTapeAttachment.sequence.status.currentStep = #JOB_2_STEP_41) AND "Unit1.Em3.ControlNodes".topTapeAttachment.sequence.status.seqActive;
   "Unit1.Em3.ControlNodes".topTapeAttachment."step".action1[241] := #_w1 AND NOT "Unit1.Em3.ControlNodes".cmTopTapeCutterUpDown.monitoring.inHomePos;
   "Unit1.Em3.ControlNodes".topTapeAttachment."step".transition1[241] := #_w1 AND "Unit1.Em3.ControlNodes".cmTopTapeCutterUpDown.monitoring.inHomePos;
   #statTonTime[241].TON(IN := #_w1 AND "Unit1.Em3.ControlNodes".topTapeAttachment."step".transition1[241],
                         PT := T#100ms);
   IF #statTonTime[241].Q THEN
       "Unit1.Em3.ControlNodes".topTapeAttachment.sequence.status.nextStep := #JOB_2_STEP_42;
   END_IF;
END_REGION

REGION Network 22: Step[242] : Top Tape Clamp Loading Open, CutterClampUp
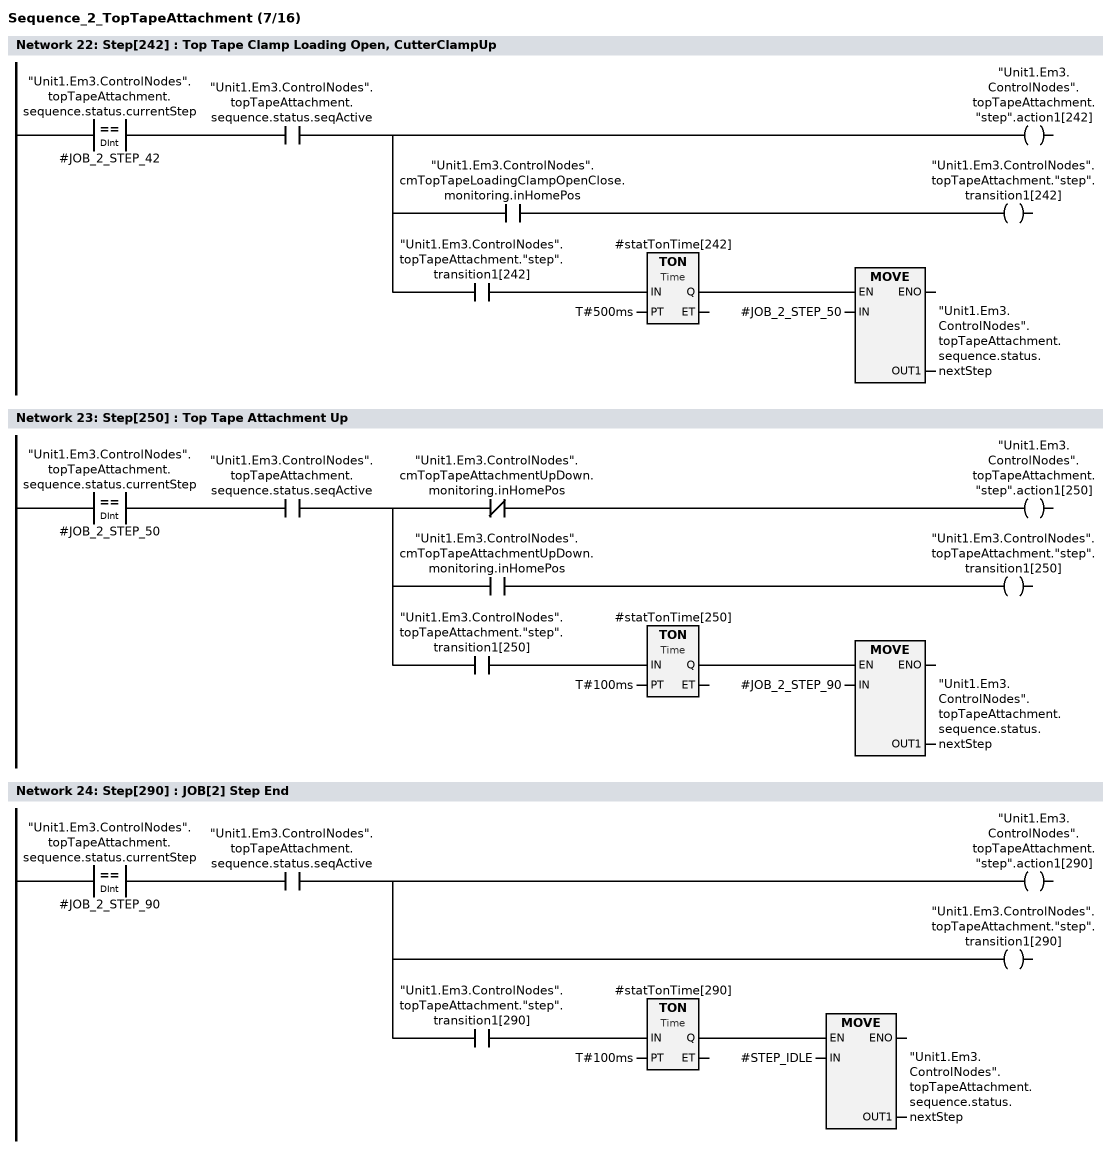
   RUNG wire#powerrail
      { S7_Templates := "SrcType := DInt" } EQ_Contact(in1 := "Unit1.Em3.ControlNodes".topTapeAttachment.sequence.status.currentStep, in2 := #JOB_2_STEP_42)
      Contact( "Unit1.Em3.ControlNodes".topTapeAttachment.sequence.status.seqActive )
      wire#w1
      Coil( "Unit1.Em3.ControlNodes".topTapeAttachment."step".action1[242] )
   END_RUNG
   RUNG wire#w1
      Contact( "Unit1.Em3.ControlNodes".cmTopTapeLoadingClampOpenClose.monitoring.inHomePos )
      Coil( "Unit1.Em3.ControlNodes".topTapeAttachment."step".transition1[242] )
   END_RUNG
   RUNG wire#w1
      Contact( "Unit1.Em3.ControlNodes".topTapeAttachment."step".transition1[242] )
      { S7_Templates := "time_type := Time" } #statTonTime[242].TON(pt := T#500ms, et =>)
      Move(in := #JOB_2_STEP_50, out1 => "Unit1.Em3.ControlNodes".topTapeAttachment.sequence.status.nextStep)
   END_RUNG
   // the same network as SCL:
   "Unit1.Em3.ControlNodes".topTapeAttachment."step".action1[242] := ("Unit1.Em3.ControlNodes".topTapeAttachment.sequence.status.currentStep = #JOB_2_STEP_42) AND "Unit1.Em3.ControlNodes".topTapeAttachment.sequence.status.seqActive;
   "Unit1.Em3.ControlNodes".topTapeAttachment."step".transition1[242] := ("Unit1.Em3.ControlNodes".topTapeAttachment.sequence.status.currentStep = #JOB_2_STEP_42) AND "Unit1.Em3.ControlNodes".topTapeAttachment.sequence.status.seqActive AND "Unit1.Em3.ControlNodes".cmTopTapeLoadingClampOpenClose.monitoring.inHomePos;
   #statTonTime[242].TON(IN := ("Unit1.Em3.ControlNodes".topTapeAttachment.sequence.status.currentStep = #JOB_2_STEP_42) AND "Unit1.Em3.ControlNodes".topTapeAttachment.sequence.status.seqActive AND "Unit1.Em3.ControlNodes".topTapeAttachment."step".transition1[242],
                         PT := T#500ms);
   IF #statTonTime[242].Q THEN
       "Unit1.Em3.ControlNodes".topTapeAttachment.sequence.status.nextStep := #JOB_2_STEP_50;
   END_IF;
END_REGION

REGION Network 23: Step[250] : Top Tape Attachment Up
   RUNG wire#powerrail
      { S7_Templates := "SrcType := DInt" } EQ_Contact(in1 := "Unit1.Em3.ControlNodes".topTapeAttachment.sequence.status.currentStep, in2 := #JOB_2_STEP_50)
      Contact( "Unit1.Em3.ControlNodes".topTapeAttachment.sequence.status.seqActive )
      wire#w1
      I_Contact( "Unit1.Em3.ControlNodes".cmTopTapeAttachmentUpDown.monitoring.inHomePos )
      Coil( "Unit1.Em3.ControlNodes".topTapeAttachment."step".action1[250] )
   END_RUNG
   RUNG wire#w1
      Contact( "Unit1.Em3.ControlNodes".cmTopTapeAttachmentUpDown.monitoring.inHomePos )
      Coil( "Unit1.Em3.ControlNodes".topTapeAttachment."step".transition1[250] )
   END_RUNG
   RUNG wire#w1
      Contact( "Unit1.Em3.ControlNodes".topTapeAttachment."step".transition1[250] )
      { S7_Templates := "time_type := Time" } #statTonTime[250].TON(pt := T#100ms, et =>)
      Move(in := #JOB_2_STEP_90, out1 => "Unit1.Em3.ControlNodes".topTapeAttachment.sequence.status.nextStep)
   END_RUNG
   // the same network as SCL:
   #_w1 := ("Unit1.Em3.ControlNodes".topTapeAttachment.sequence.status.currentStep = #JOB_2_STEP_50) AND "Unit1.Em3.ControlNodes".topTapeAttachment.sequence.status.seqActive;
   "Unit1.Em3.ControlNodes".topTapeAttachment."step".action1[250] := #_w1 AND NOT "Unit1.Em3.ControlNodes".cmTopTapeAttachmentUpDown.monitoring.inHomePos;
   "Unit1.Em3.ControlNodes".topTapeAttachment."step".transition1[250] := #_w1 AND "Unit1.Em3.ControlNodes".cmTopTapeAttachmentUpDown.monitoring.inHomePos;
   #statTonTime[250].TON(IN := #_w1 AND "Unit1.Em3.ControlNodes".topTapeAttachment."step".transition1[250],
                         PT := T#100ms);
   IF #statTonTime[250].Q THEN
       "Unit1.Em3.ControlNodes".topTapeAttachment.sequence.status.nextStep := #JOB_2_STEP_90;
   END_IF;
END_REGION

REGION Network 24: Step[290] : JOB[2] Step End
   RUNG wire#powerrail
      { S7_Templates := "SrcType := DInt" } EQ_Contact(in1 := "Unit1.Em3.ControlNodes".topTapeAttachment.sequence.status.currentStep, in2 := #JOB_2_STEP_90)
      Contact( "Unit1.Em3.ControlNodes".topTapeAttachment.sequence.status.seqActive )
      wire#w1
      Coil( "Unit1.Em3.ControlNodes".topTapeAttachment."step".action1[290] )
   END_RUNG
   RUNG wire#w1
      Coil( "Unit1.Em3.ControlNodes".topTapeAttachment."step".transition1[290] )
   END_RUNG
   RUNG wire#w1
      Contact( "Unit1.Em3.ControlNodes".topTapeAttachment."step".transition1[290] )
      { S7_Templates := "time_type := Time" } #statTonTime[290].TON(pt := T#100ms, et =>)
      Move(in := #STEP_IDLE, out1 => "Unit1.Em3.ControlNodes".topTapeAttachment.sequence.status.nextStep)
   END_RUNG
   // the same network as SCL:
   "Unit1.Em3.ControlNodes".topTapeAttachment."step".action1[290] := ("Unit1.Em3.ControlNodes".topTapeAttachment.sequence.status.currentStep = #JOB_2_STEP_90) AND "Unit1.Em3.ControlNodes".topTapeAttachment.sequence.status.seqActive;
   "Unit1.Em3.ControlNodes".topTapeAttachment."step".transition1[290] := ("Unit1.Em3.ControlNodes".topTapeAttachment.sequence.status.currentStep = #JOB_2_STEP_90) AND "Unit1.Em3.ControlNodes".topTapeAttachment.sequence.status.seqActive;
   #statTonTime[290].TON(IN := ("Unit1.Em3.ControlNodes".topTapeAttachment.sequence.status.currentStep = #JOB_2_STEP_90) AND "Unit1.Em3.ControlNodes".topTapeAttachment.sequence.status.seqActive AND "Unit1.Em3.ControlNodes".topTapeAttachment."step".transition1[290],
                         PT := T#100ms);
   IF #statTonTime[290].Q THEN
       "Unit1.Em3.ControlNodes".topTapeAttachment.sequence.status.nextStep := #STEP_IDLE;
   END_IF;
END_REGION

REGION Network 25: *************** JOB[3] TOP TAPE PUT-1=AUTO *************************
END_REGION

REGION Network 26: Step[301] : JOB[3] Condition
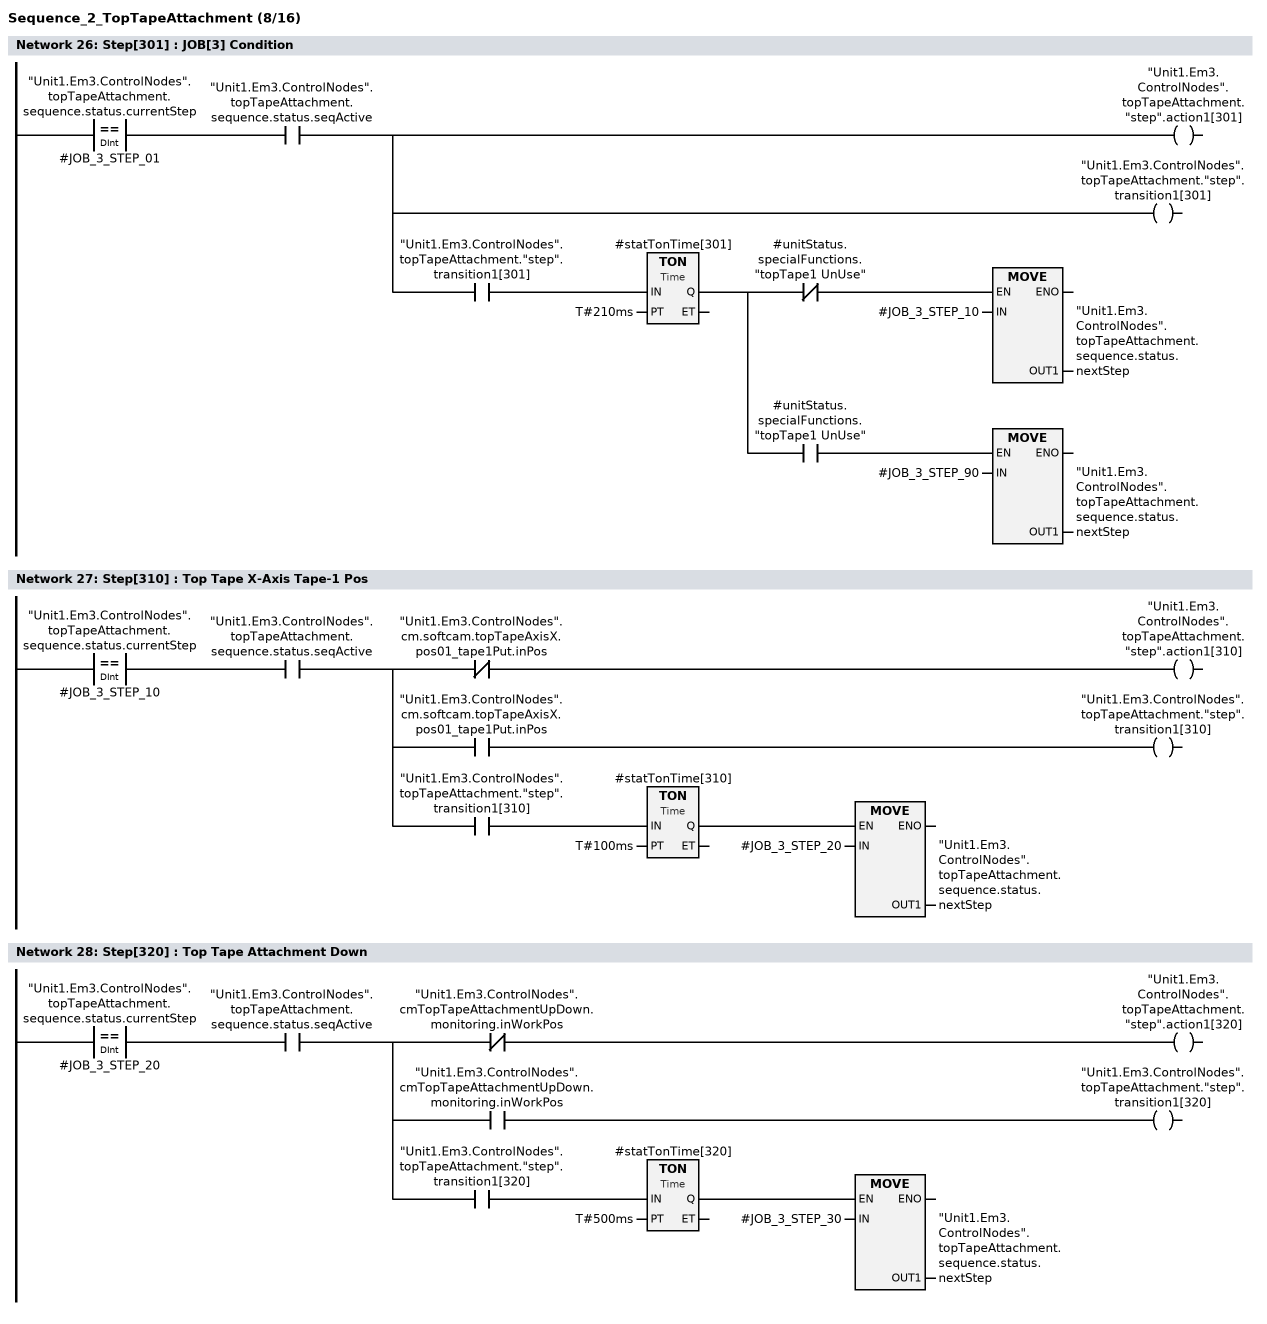
   RUNG wire#powerrail
      { S7_Templates := "SrcType := DInt" } EQ_Contact(in1 := "Unit1.Em3.ControlNodes".topTapeAttachment.sequence.status.currentStep, in2 := #JOB_3_STEP_01)
      Contact( "Unit1.Em3.ControlNodes".topTapeAttachment.sequence.status.seqActive )
      wire#w1
      Coil( "Unit1.Em3.ControlNodes".topTapeAttachment."step".action1[301] )
   END_RUNG
   RUNG wire#w1
      Coil( "Unit1.Em3.ControlNodes".topTapeAttachment."step".transition1[301] )
   END_RUNG
   RUNG wire#w1
      Contact( "Unit1.Em3.ControlNodes".topTapeAttachment."step".transition1[301] )
      { S7_Templates := "time_type := Time" } #statTonTime[301].TON(pt := T#210ms, et =>)
      wire#w2
      I_Contact( #unitStatus.specialFunctions."topTape1 UnUse" )
      Move(in := #JOB_3_STEP_10, out1 => "Unit1.Em3.ControlNodes".topTapeAttachment.sequence.status.nextStep)
   END_RUNG
   RUNG wire#w2
      Contact( #unitStatus.specialFunctions."topTape1 UnUse" )
      Move(in := #JOB_3_STEP_90, out1 => "Unit1.Em3.ControlNodes".topTapeAttachment.sequence.status.nextStep)
   END_RUNG
   // the same network as SCL:
   "Unit1.Em3.ControlNodes".topTapeAttachment."step".action1[301] := ("Unit1.Em3.ControlNodes".topTapeAttachment.sequence.status.currentStep = #JOB_3_STEP_01) AND "Unit1.Em3.ControlNodes".topTapeAttachment.sequence.status.seqActive;
   "Unit1.Em3.ControlNodes".topTapeAttachment."step".transition1[301] := ("Unit1.Em3.ControlNodes".topTapeAttachment.sequence.status.currentStep = #JOB_3_STEP_01) AND "Unit1.Em3.ControlNodes".topTapeAttachment.sequence.status.seqActive;
   #statTonTime[301].TON(IN := ("Unit1.Em3.ControlNodes".topTapeAttachment.sequence.status.currentStep = #JOB_3_STEP_01) AND "Unit1.Em3.ControlNodes".topTapeAttachment.sequence.status.seqActive AND "Unit1.Em3.ControlNodes".topTapeAttachment."step".transition1[301],
                         PT := T#210ms);
   IF #statTonTime[301].Q AND NOT #unitStatus.specialFunctions."topTape1 UnUse" THEN
       "Unit1.Em3.ControlNodes".topTapeAttachment.sequence.status.nextStep := #JOB_3_STEP_10;
   END_IF;
   IF #statTonTime[301].Q AND #unitStatus.specialFunctions."topTape1 UnUse" THEN
       "Unit1.Em3.ControlNodes".topTapeAttachment.sequence.status.nextStep := #JOB_3_STEP_90;
   END_IF;
END_REGION

REGION Network 27: Step[310] : Top Tape X-Axis Tape-1 Pos
   RUNG wire#powerrail
      { S7_Templates := "SrcType := DInt" } EQ_Contact(in1 := "Unit1.Em3.ControlNodes".topTapeAttachment.sequence.status.currentStep, in2 := #JOB_3_STEP_10)
      Contact( "Unit1.Em3.ControlNodes".topTapeAttachment.sequence.status.seqActive )
      wire#w1
      I_Contact( "Unit1.Em3.ControlNodes".cm.softcam.topTapeAxisX.pos01_tape1Put.inPos )
      Coil( "Unit1.Em3.ControlNodes".topTapeAttachment."step".action1[310] )
   END_RUNG
   RUNG wire#w1
      Contact( "Unit1.Em3.ControlNodes".cm.softcam.topTapeAxisX.pos01_tape1Put.inPos )
      Coil( "Unit1.Em3.ControlNodes".topTapeAttachment."step".transition1[310] )
   END_RUNG
   RUNG wire#w1
      Contact( "Unit1.Em3.ControlNodes".topTapeAttachment."step".transition1[310] )
      { S7_Templates := "time_type := Time" } #statTonTime[310].TON(pt := T#100ms, et =>)
      Move(in := #JOB_3_STEP_20, out1 => "Unit1.Em3.ControlNodes".topTapeAttachment.sequence.status.nextStep)
   END_RUNG
   // the same network as SCL:
   #_w1 := ("Unit1.Em3.ControlNodes".topTapeAttachment.sequence.status.currentStep = #JOB_3_STEP_10) AND "Unit1.Em3.ControlNodes".topTapeAttachment.sequence.status.seqActive;
   "Unit1.Em3.ControlNodes".topTapeAttachment."step".action1[310] := #_w1 AND NOT "Unit1.Em3.ControlNodes".cm.softcam.topTapeAxisX.pos01_tape1Put.inPos;
   "Unit1.Em3.ControlNodes".topTapeAttachment."step".transition1[310] := #_w1 AND "Unit1.Em3.ControlNodes".cm.softcam.topTapeAxisX.pos01_tape1Put.inPos;
   #statTonTime[310].TON(IN := #_w1 AND "Unit1.Em3.ControlNodes".topTapeAttachment."step".transition1[310],
                         PT := T#100ms);
   IF #statTonTime[310].Q THEN
       "Unit1.Em3.ControlNodes".topTapeAttachment.sequence.status.nextStep := #JOB_3_STEP_20;
   END_IF;
END_REGION

REGION Network 28: Step[320] : Top Tape Attachment Down
   RUNG wire#powerrail
      { S7_Templates := "SrcType := DInt" } EQ_Contact(in1 := "Unit1.Em3.ControlNodes".topTapeAttachment.sequence.status.currentStep, in2 := #JOB_3_STEP_20)
      Contact( "Unit1.Em3.ControlNodes".topTapeAttachment.sequence.status.seqActive )
      wire#w1
      I_Contact( "Unit1.Em3.ControlNodes".cmTopTapeAttachmentUpDown.monitoring.inWorkPos )
      Coil( "Unit1.Em3.ControlNodes".topTapeAttachment."step".action1[320] )
   END_RUNG
   RUNG wire#w1
      Contact( "Unit1.Em3.ControlNodes".cmTopTapeAttachmentUpDown.monitoring.inWorkPos )
      Coil( "Unit1.Em3.ControlNodes".topTapeAttachment."step".transition1[320] )
   END_RUNG
   RUNG wire#w1
      Contact( "Unit1.Em3.ControlNodes".topTapeAttachment."step".transition1[320] )
      { S7_Templates := "time_type := Time" } #statTonTime[320].TON(pt := T#500ms, et =>)
      Move(in := #JOB_3_STEP_30, out1 => "Unit1.Em3.ControlNodes".topTapeAttachment.sequence.status.nextStep)
   END_RUNG
   // the same network as SCL:
   #_w1 := ("Unit1.Em3.ControlNodes".topTapeAttachment.sequence.status.currentStep = #JOB_3_STEP_20) AND "Unit1.Em3.ControlNodes".topTapeAttachment.sequence.status.seqActive;
   "Unit1.Em3.ControlNodes".topTapeAttachment."step".action1[320] := #_w1 AND NOT "Unit1.Em3.ControlNodes".cmTopTapeAttachmentUpDown.monitoring.inWorkPos;
   "Unit1.Em3.ControlNodes".topTapeAttachment."step".transition1[320] := #_w1 AND "Unit1.Em3.ControlNodes".cmTopTapeAttachmentUpDown.monitoring.inWorkPos;
   #statTonTime[320].TON(IN := #_w1 AND "Unit1.Em3.ControlNodes".topTapeAttachment."step".transition1[320],
                         PT := T#500ms);
   IF #statTonTime[320].Q THEN
       "Unit1.Em3.ControlNodes".topTapeAttachment.sequence.status.nextStep := #JOB_3_STEP_30;
   END_IF;
END_REGION

REGION Network 29: Step[330] : Top Tape Attachment Vaccum Off
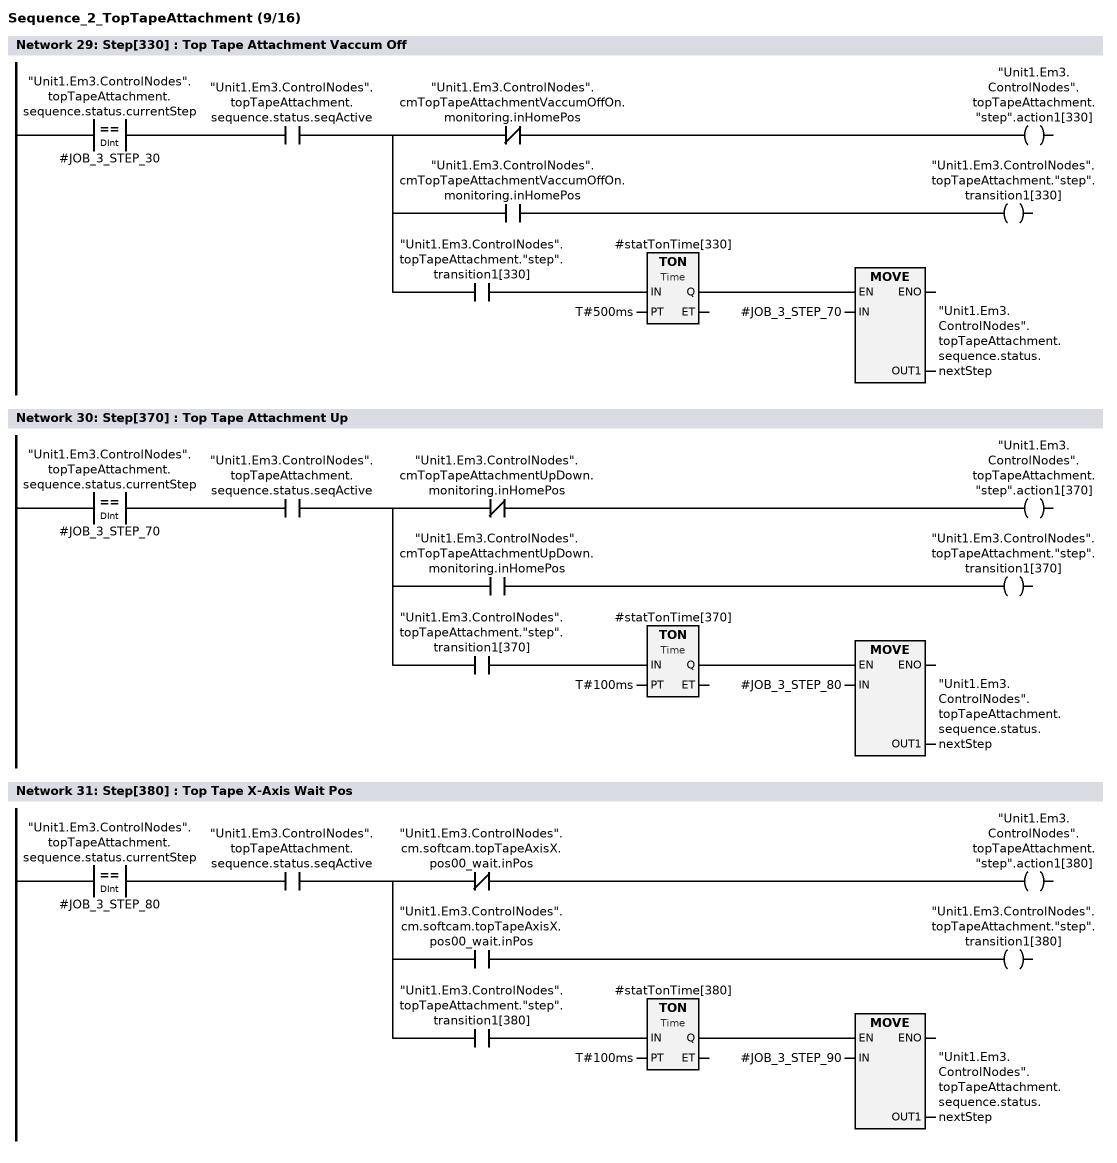
   RUNG wire#powerrail
      { S7_Templates := "SrcType := DInt" } EQ_Contact(in1 := "Unit1.Em3.ControlNodes".topTapeAttachment.sequence.status.currentStep, in2 := #JOB_3_STEP_30)
      Contact( "Unit1.Em3.ControlNodes".topTapeAttachment.sequence.status.seqActive )
      wire#w1
      I_Contact( "Unit1.Em3.ControlNodes".cmTopTapeAttachmentVaccumOffOn.monitoring.inHomePos )
      Coil( "Unit1.Em3.ControlNodes".topTapeAttachment."step".action1[330] )
   END_RUNG
   RUNG wire#w1
      Contact( "Unit1.Em3.ControlNodes".cmTopTapeAttachmentVaccumOffOn.monitoring.inHomePos )
      Coil( "Unit1.Em3.ControlNodes".topTapeAttachment."step".transition1[330] )
   END_RUNG
   RUNG wire#w1
      Contact( "Unit1.Em3.ControlNodes".topTapeAttachment."step".transition1[330] )
      { S7_Templates := "time_type := Time" } #statTonTime[330].TON(pt := T#500ms, et =>)
      Move(in := #JOB_3_STEP_70, out1 => "Unit1.Em3.ControlNodes".topTapeAttachment.sequence.status.nextStep)
   END_RUNG
   // the same network as SCL:
   #_w1 := ("Unit1.Em3.ControlNodes".topTapeAttachment.sequence.status.currentStep = #JOB_3_STEP_30) AND "Unit1.Em3.ControlNodes".topTapeAttachment.sequence.status.seqActive;
   "Unit1.Em3.ControlNodes".topTapeAttachment."step".action1[330] := #_w1 AND NOT "Unit1.Em3.ControlNodes".cmTopTapeAttachmentVaccumOffOn.monitoring.inHomePos;
   "Unit1.Em3.ControlNodes".topTapeAttachment."step".transition1[330] := #_w1 AND "Unit1.Em3.ControlNodes".cmTopTapeAttachmentVaccumOffOn.monitoring.inHomePos;
   #statTonTime[330].TON(IN := #_w1 AND "Unit1.Em3.ControlNodes".topTapeAttachment."step".transition1[330],
                         PT := T#500ms);
   IF #statTonTime[330].Q THEN
       "Unit1.Em3.ControlNodes".topTapeAttachment.sequence.status.nextStep := #JOB_3_STEP_70;
   END_IF;
END_REGION

REGION Network 30: Step[370] : Top Tape Attachment Up
   RUNG wire#powerrail
      { S7_Templates := "SrcType := DInt" } EQ_Contact(in1 := "Unit1.Em3.ControlNodes".topTapeAttachment.sequence.status.currentStep, in2 := #JOB_3_STEP_70)
      Contact( "Unit1.Em3.ControlNodes".topTapeAttachment.sequence.status.seqActive )
      wire#w1
      I_Contact( "Unit1.Em3.ControlNodes".cmTopTapeAttachmentUpDown.monitoring.inHomePos )
      Coil( "Unit1.Em3.ControlNodes".topTapeAttachment."step".action1[370] )
   END_RUNG
   RUNG wire#w1
      Contact( "Unit1.Em3.ControlNodes".cmTopTapeAttachmentUpDown.monitoring.inHomePos )
      Coil( "Unit1.Em3.ControlNodes".topTapeAttachment."step".transition1[370] )
   END_RUNG
   RUNG wire#w1
      Contact( "Unit1.Em3.ControlNodes".topTapeAttachment."step".transition1[370] )
      { S7_Templates := "time_type := Time" } #statTonTime[370].TON(pt := T#100ms, et =>)
      Move(in := #JOB_3_STEP_80, out1 => "Unit1.Em3.ControlNodes".topTapeAttachment.sequence.status.nextStep)
   END_RUNG
   // the same network as SCL:
   #_w1 := ("Unit1.Em3.ControlNodes".topTapeAttachment.sequence.status.currentStep = #JOB_3_STEP_70) AND "Unit1.Em3.ControlNodes".topTapeAttachment.sequence.status.seqActive;
   "Unit1.Em3.ControlNodes".topTapeAttachment."step".action1[370] := #_w1 AND NOT "Unit1.Em3.ControlNodes".cmTopTapeAttachmentUpDown.monitoring.inHomePos;
   "Unit1.Em3.ControlNodes".topTapeAttachment."step".transition1[370] := #_w1 AND "Unit1.Em3.ControlNodes".cmTopTapeAttachmentUpDown.monitoring.inHomePos;
   #statTonTime[370].TON(IN := #_w1 AND "Unit1.Em3.ControlNodes".topTapeAttachment."step".transition1[370],
                         PT := T#100ms);
   IF #statTonTime[370].Q THEN
       "Unit1.Em3.ControlNodes".topTapeAttachment.sequence.status.nextStep := #JOB_3_STEP_80;
   END_IF;
END_REGION

REGION Network 31: Step[380] : Top Tape X-Axis Wait Pos
   RUNG wire#powerrail
      { S7_Templates := "SrcType := DInt" } EQ_Contact(in1 := "Unit1.Em3.ControlNodes".topTapeAttachment.sequence.status.currentStep, in2 := #JOB_3_STEP_80)
      Contact( "Unit1.Em3.ControlNodes".topTapeAttachment.sequence.status.seqActive )
      wire#w1
      I_Contact( "Unit1.Em3.ControlNodes".cm.softcam.topTapeAxisX.pos00_wait.inPos )
      Coil( "Unit1.Em3.ControlNodes".topTapeAttachment."step".action1[380] )
   END_RUNG
   RUNG wire#w1
      Contact( "Unit1.Em3.ControlNodes".cm.softcam.topTapeAxisX.pos00_wait.inPos )
      Coil( "Unit1.Em3.ControlNodes".topTapeAttachment."step".transition1[380] )
   END_RUNG
   RUNG wire#w1
      Contact( "Unit1.Em3.ControlNodes".topTapeAttachment."step".transition1[380] )
      { S7_Templates := "time_type := Time" } #statTonTime[380].TON(pt := T#100ms, et =>)
      Move(in := #JOB_3_STEP_90, out1 => "Unit1.Em3.ControlNodes".topTapeAttachment.sequence.status.nextStep)
   END_RUNG
   // the same network as SCL:
   #_w1 := ("Unit1.Em3.ControlNodes".topTapeAttachment.sequence.status.currentStep = #JOB_3_STEP_80) AND "Unit1.Em3.ControlNodes".topTapeAttachment.sequence.status.seqActive;
   "Unit1.Em3.ControlNodes".topTapeAttachment."step".action1[380] := #_w1 AND NOT "Unit1.Em3.ControlNodes".cm.softcam.topTapeAxisX.pos00_wait.inPos;
   "Unit1.Em3.ControlNodes".topTapeAttachment."step".transition1[380] := #_w1 AND "Unit1.Em3.ControlNodes".cm.softcam.topTapeAxisX.pos00_wait.inPos;
   #statTonTime[380].TON(IN := #_w1 AND "Unit1.Em3.ControlNodes".topTapeAttachment."step".transition1[380],
                         PT := T#100ms);
   IF #statTonTime[380].Q THEN
       "Unit1.Em3.ControlNodes".topTapeAttachment.sequence.status.nextStep := #JOB_3_STEP_90;
   END_IF;
END_REGION

REGION Network 32: Step[390] : JOB[3] Step End
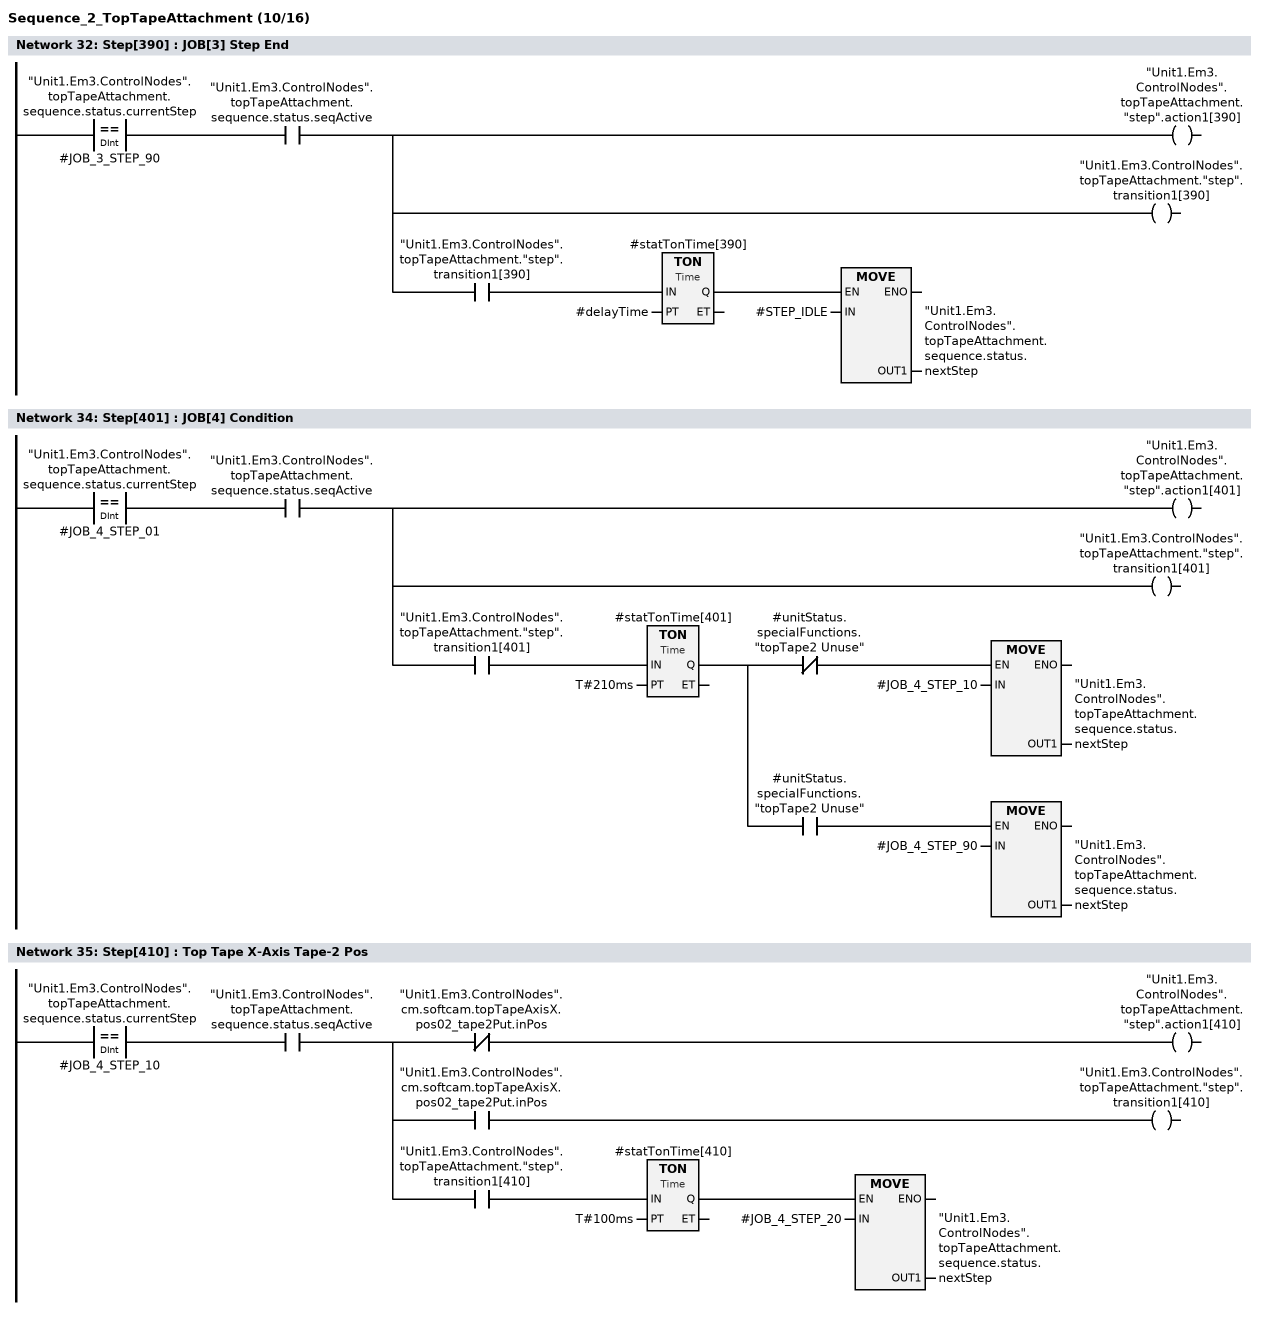
   RUNG wire#powerrail
      { S7_Templates := "SrcType := DInt" } EQ_Contact(in1 := "Unit1.Em3.ControlNodes".topTapeAttachment.sequence.status.currentStep, in2 := #JOB_3_STEP_90)
      Contact( "Unit1.Em3.ControlNodes".topTapeAttachment.sequence.status.seqActive )
      wire#w1
      Coil( "Unit1.Em3.ControlNodes".topTapeAttachment."step".action1[390] )
   END_RUNG
   RUNG wire#w1
      Coil( "Unit1.Em3.ControlNodes".topTapeAttachment."step".transition1[390] )
   END_RUNG
   RUNG wire#w1
      Contact( "Unit1.Em3.ControlNodes".topTapeAttachment."step".transition1[390] )
      { S7_Templates := "time_type := Time" } #statTonTime[390].TON(pt := #delayTime, et =>)
      Move(in := #STEP_IDLE, out1 => "Unit1.Em3.ControlNodes".topTapeAttachment.sequence.status.nextStep)
   END_RUNG
   // the same network as SCL:
   "Unit1.Em3.ControlNodes".topTapeAttachment."step".action1[390] := ("Unit1.Em3.ControlNodes".topTapeAttachment.sequence.status.currentStep = #JOB_3_STEP_90) AND "Unit1.Em3.ControlNodes".topTapeAttachment.sequence.status.seqActive;
   "Unit1.Em3.ControlNodes".topTapeAttachment."step".transition1[390] := ("Unit1.Em3.ControlNodes".topTapeAttachment.sequence.status.currentStep = #JOB_3_STEP_90) AND "Unit1.Em3.ControlNodes".topTapeAttachment.sequence.status.seqActive;
   #statTonTime[390].TON(IN := ("Unit1.Em3.ControlNodes".topTapeAttachment.sequence.status.currentStep = #JOB_3_STEP_90) AND "Unit1.Em3.ControlNodes".topTapeAttachment.sequence.status.seqActive AND "Unit1.Em3.ControlNodes".topTapeAttachment."step".transition1[390],
                         PT := #delayTime);
   IF #statTonTime[390].Q THEN
       "Unit1.Em3.ControlNodes".topTapeAttachment.sequence.status.nextStep := #STEP_IDLE;
   END_IF;
END_REGION

REGION Network 33: *************** JOB[4] TOP TAPE PUT-2=AUTO *************************
END_REGION

REGION Network 34: Step[401] : JOB[4] Condition
   RUNG wire#powerrail
      { S7_Templates := "SrcType := DInt" } EQ_Contact(in1 := "Unit1.Em3.ControlNodes".topTapeAttachment.sequence.status.currentStep, in2 := #JOB_4_STEP_01)
      Contact( "Unit1.Em3.ControlNodes".topTapeAttachment.sequence.status.seqActive )
      wire#w1
      Coil( "Unit1.Em3.ControlNodes".topTapeAttachment."step".action1[401] )
   END_RUNG
   RUNG wire#w1
      Coil( "Unit1.Em3.ControlNodes".topTapeAttachment."step".transition1[401] )
   END_RUNG
   RUNG wire#w1
      Contact( "Unit1.Em3.ControlNodes".topTapeAttachment."step".transition1[401] )
      { S7_Templates := "time_type := Time" } #statTonTime[401].TON(pt := T#210ms, et =>)
      wire#w2
      I_Contact( #unitStatus.specialFunctions."topTape2 Unuse" )
      Move(in := #JOB_4_STEP_10, out1 => "Unit1.Em3.ControlNodes".topTapeAttachment.sequence.status.nextStep)
   END_RUNG
   RUNG wire#w2
      Contact( #unitStatus.specialFunctions."topTape2 Unuse" )
      Move(in := #JOB_4_STEP_90, out1 => "Unit1.Em3.ControlNodes".topTapeAttachment.sequence.status.nextStep)
   END_RUNG
   // the same network as SCL:
   "Unit1.Em3.ControlNodes".topTapeAttachment."step".action1[401] := ("Unit1.Em3.ControlNodes".topTapeAttachment.sequence.status.currentStep = #JOB_4_STEP_01) AND "Unit1.Em3.ControlNodes".topTapeAttachment.sequence.status.seqActive;
   "Unit1.Em3.ControlNodes".topTapeAttachment."step".transition1[401] := ("Unit1.Em3.ControlNodes".topTapeAttachment.sequence.status.currentStep = #JOB_4_STEP_01) AND "Unit1.Em3.ControlNodes".topTapeAttachment.sequence.status.seqActive;
   #statTonTime[401].TON(IN := ("Unit1.Em3.ControlNodes".topTapeAttachment.sequence.status.currentStep = #JOB_4_STEP_01) AND "Unit1.Em3.ControlNodes".topTapeAttachment.sequence.status.seqActive AND "Unit1.Em3.ControlNodes".topTapeAttachment."step".transition1[401],
                         PT := T#210ms);
   IF #statTonTime[401].Q AND NOT #unitStatus.specialFunctions."topTape2 Unuse" THEN
       "Unit1.Em3.ControlNodes".topTapeAttachment.sequence.status.nextStep := #JOB_4_STEP_10;
   END_IF;
   IF #statTonTime[401].Q AND #unitStatus.specialFunctions."topTape2 Unuse" THEN
       "Unit1.Em3.ControlNodes".topTapeAttachment.sequence.status.nextStep := #JOB_4_STEP_90;
   END_IF;
END_REGION

REGION Network 35: Step[410] : Top Tape X-Axis Tape-2 Pos
   RUNG wire#powerrail
      { S7_Templates := "SrcType := DInt" } EQ_Contact(in1 := "Unit1.Em3.ControlNodes".topTapeAttachment.sequence.status.currentStep, in2 := #JOB_4_STEP_10)
      Contact( "Unit1.Em3.ControlNodes".topTapeAttachment.sequence.status.seqActive )
      wire#w1
      I_Contact( "Unit1.Em3.ControlNodes".cm.softcam.topTapeAxisX.pos02_tape2Put.inPos )
      Coil( "Unit1.Em3.ControlNodes".topTapeAttachment."step".action1[410] )
   END_RUNG
   RUNG wire#w1
      Contact( "Unit1.Em3.ControlNodes".cm.softcam.topTapeAxisX.pos02_tape2Put.inPos )
      Coil( "Unit1.Em3.ControlNodes".topTapeAttachment."step".transition1[410] )
   END_RUNG
   RUNG wire#w1
      Contact( "Unit1.Em3.ControlNodes".topTapeAttachment."step".transition1[410] )
      { S7_Templates := "time_type := Time" } #statTonTime[410].TON(pt := T#100ms, et =>)
      Move(in := #JOB_4_STEP_20, out1 => "Unit1.Em3.ControlNodes".topTapeAttachment.sequence.status.nextStep)
   END_RUNG
   // the same network as SCL:
   #_w1 := ("Unit1.Em3.ControlNodes".topTapeAttachment.sequence.status.currentStep = #JOB_4_STEP_10) AND "Unit1.Em3.ControlNodes".topTapeAttachment.sequence.status.seqActive;
   "Unit1.Em3.ControlNodes".topTapeAttachment."step".action1[410] := #_w1 AND NOT "Unit1.Em3.ControlNodes".cm.softcam.topTapeAxisX.pos02_tape2Put.inPos;
   "Unit1.Em3.ControlNodes".topTapeAttachment."step".transition1[410] := #_w1 AND "Unit1.Em3.ControlNodes".cm.softcam.topTapeAxisX.pos02_tape2Put.inPos;
   #statTonTime[410].TON(IN := #_w1 AND "Unit1.Em3.ControlNodes".topTapeAttachment."step".transition1[410],
                         PT := T#100ms);
   IF #statTonTime[410].Q THEN
       "Unit1.Em3.ControlNodes".topTapeAttachment.sequence.status.nextStep := #JOB_4_STEP_20;
   END_IF;
END_REGION

REGION Network 36: Step[420] : Top Tape Attachment Down
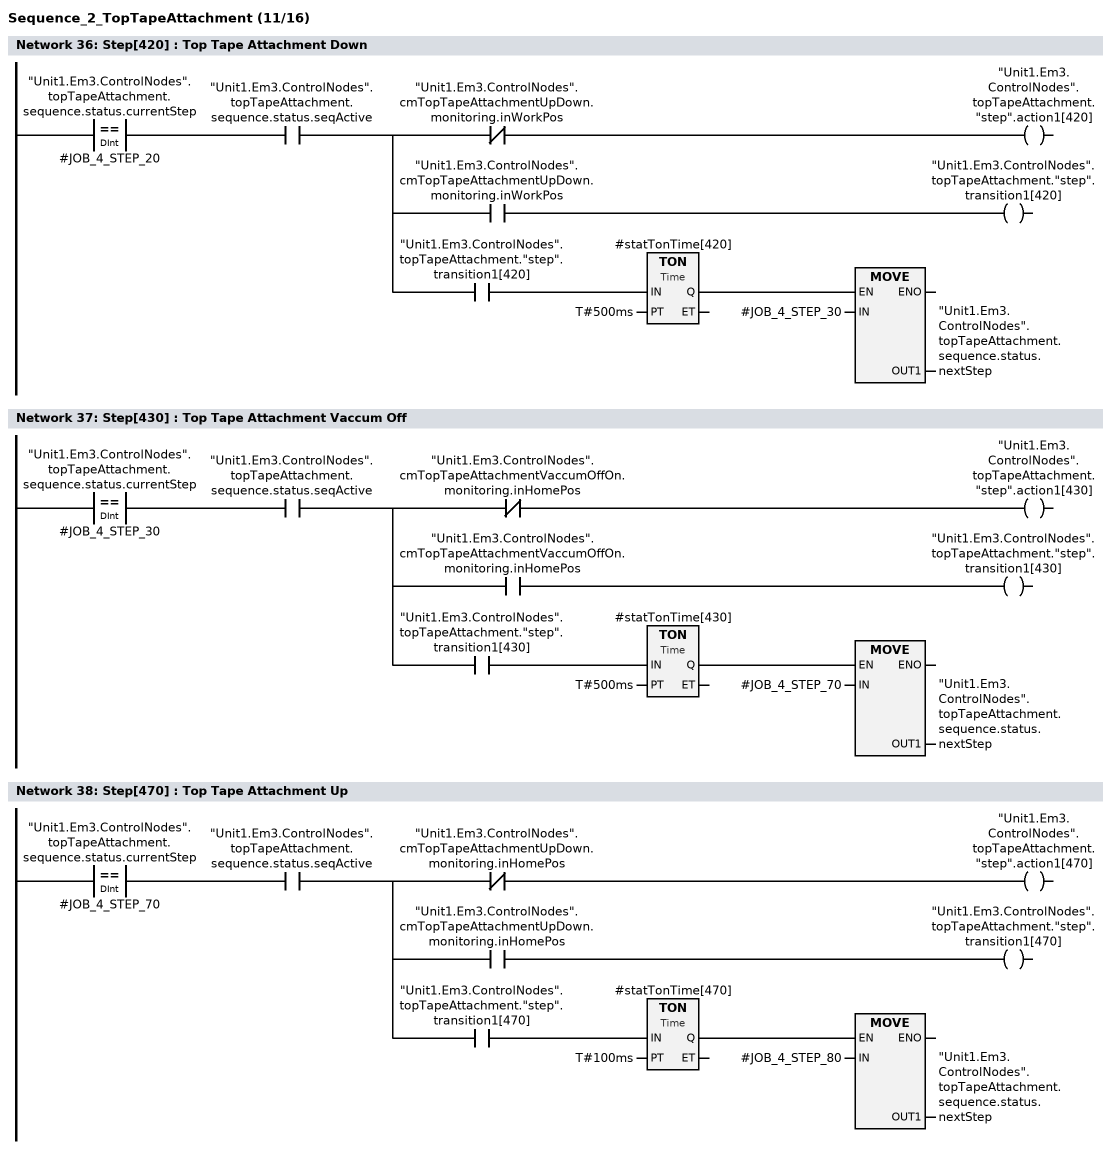
   RUNG wire#powerrail
      { S7_Templates := "SrcType := DInt" } EQ_Contact(in1 := "Unit1.Em3.ControlNodes".topTapeAttachment.sequence.status.currentStep, in2 := #JOB_4_STEP_20)
      Contact( "Unit1.Em3.ControlNodes".topTapeAttachment.sequence.status.seqActive )
      wire#w1
      I_Contact( "Unit1.Em3.ControlNodes".cmTopTapeAttachmentUpDown.monitoring.inWorkPos )
      Coil( "Unit1.Em3.ControlNodes".topTapeAttachment."step".action1[420] )
   END_RUNG
   RUNG wire#w1
      Contact( "Unit1.Em3.ControlNodes".cmTopTapeAttachmentUpDown.monitoring.inWorkPos )
      Coil( "Unit1.Em3.ControlNodes".topTapeAttachment."step".transition1[420] )
   END_RUNG
   RUNG wire#w1
      Contact( "Unit1.Em3.ControlNodes".topTapeAttachment."step".transition1[420] )
      { S7_Templates := "time_type := Time" } #statTonTime[420].TON(pt := T#500ms, et =>)
      Move(in := #JOB_4_STEP_30, out1 => "Unit1.Em3.ControlNodes".topTapeAttachment.sequence.status.nextStep)
   END_RUNG
   // the same network as SCL:
   #_w1 := ("Unit1.Em3.ControlNodes".topTapeAttachment.sequence.status.currentStep = #JOB_4_STEP_20) AND "Unit1.Em3.ControlNodes".topTapeAttachment.sequence.status.seqActive;
   "Unit1.Em3.ControlNodes".topTapeAttachment."step".action1[420] := #_w1 AND NOT "Unit1.Em3.ControlNodes".cmTopTapeAttachmentUpDown.monitoring.inWorkPos;
   "Unit1.Em3.ControlNodes".topTapeAttachment."step".transition1[420] := #_w1 AND "Unit1.Em3.ControlNodes".cmTopTapeAttachmentUpDown.monitoring.inWorkPos;
   #statTonTime[420].TON(IN := #_w1 AND "Unit1.Em3.ControlNodes".topTapeAttachment."step".transition1[420],
                         PT := T#500ms);
   IF #statTonTime[420].Q THEN
       "Unit1.Em3.ControlNodes".topTapeAttachment.sequence.status.nextStep := #JOB_4_STEP_30;
   END_IF;
END_REGION

REGION Network 37: Step[430] : Top Tape Attachment Vaccum Off
   RUNG wire#powerrail
      { S7_Templates := "SrcType := DInt" } EQ_Contact(in1 := "Unit1.Em3.ControlNodes".topTapeAttachment.sequence.status.currentStep, in2 := #JOB_4_STEP_30)
      Contact( "Unit1.Em3.ControlNodes".topTapeAttachment.sequence.status.seqActive )
      wire#w1
      I_Contact( "Unit1.Em3.ControlNodes".cmTopTapeAttachmentVaccumOffOn.monitoring.inHomePos )
      Coil( "Unit1.Em3.ControlNodes".topTapeAttachment."step".action1[430] )
   END_RUNG
   RUNG wire#w1
      Contact( "Unit1.Em3.ControlNodes".cmTopTapeAttachmentVaccumOffOn.monitoring.inHomePos )
      Coil( "Unit1.Em3.ControlNodes".topTapeAttachment."step".transition1[430] )
   END_RUNG
   RUNG wire#w1
      Contact( "Unit1.Em3.ControlNodes".topTapeAttachment."step".transition1[430] )
      { S7_Templates := "time_type := Time" } #statTonTime[430].TON(pt := T#500ms, et =>)
      Move(in := #JOB_4_STEP_70, out1 => "Unit1.Em3.ControlNodes".topTapeAttachment.sequence.status.nextStep)
   END_RUNG
   // the same network as SCL:
   #_w1 := ("Unit1.Em3.ControlNodes".topTapeAttachment.sequence.status.currentStep = #JOB_4_STEP_30) AND "Unit1.Em3.ControlNodes".topTapeAttachment.sequence.status.seqActive;
   "Unit1.Em3.ControlNodes".topTapeAttachment."step".action1[430] := #_w1 AND NOT "Unit1.Em3.ControlNodes".cmTopTapeAttachmentVaccumOffOn.monitoring.inHomePos;
   "Unit1.Em3.ControlNodes".topTapeAttachment."step".transition1[430] := #_w1 AND "Unit1.Em3.ControlNodes".cmTopTapeAttachmentVaccumOffOn.monitoring.inHomePos;
   #statTonTime[430].TON(IN := #_w1 AND "Unit1.Em3.ControlNodes".topTapeAttachment."step".transition1[430],
                         PT := T#500ms);
   IF #statTonTime[430].Q THEN
       "Unit1.Em3.ControlNodes".topTapeAttachment.sequence.status.nextStep := #JOB_4_STEP_70;
   END_IF;
END_REGION

REGION Network 38: Step[470] : Top Tape Attachment Up
   RUNG wire#powerrail
      { S7_Templates := "SrcType := DInt" } EQ_Contact(in1 := "Unit1.Em3.ControlNodes".topTapeAttachment.sequence.status.currentStep, in2 := #JOB_4_STEP_70)
      Contact( "Unit1.Em3.ControlNodes".topTapeAttachment.sequence.status.seqActive )
      wire#w1
      I_Contact( "Unit1.Em3.ControlNodes".cmTopTapeAttachmentUpDown.monitoring.inHomePos )
      Coil( "Unit1.Em3.ControlNodes".topTapeAttachment."step".action1[470] )
   END_RUNG
   RUNG wire#w1
      Contact( "Unit1.Em3.ControlNodes".cmTopTapeAttachmentUpDown.monitoring.inHomePos )
      Coil( "Unit1.Em3.ControlNodes".topTapeAttachment."step".transition1[470] )
   END_RUNG
   RUNG wire#w1
      Contact( "Unit1.Em3.ControlNodes".topTapeAttachment."step".transition1[470] )
      { S7_Templates := "time_type := Time" } #statTonTime[470].TON(pt := T#100ms, et =>)
      Move(in := #JOB_4_STEP_80, out1 => "Unit1.Em3.ControlNodes".topTapeAttachment.sequence.status.nextStep)
   END_RUNG
   // the same network as SCL:
   #_w1 := ("Unit1.Em3.ControlNodes".topTapeAttachment.sequence.status.currentStep = #JOB_4_STEP_70) AND "Unit1.Em3.ControlNodes".topTapeAttachment.sequence.status.seqActive;
   "Unit1.Em3.ControlNodes".topTapeAttachment."step".action1[470] := #_w1 AND NOT "Unit1.Em3.ControlNodes".cmTopTapeAttachmentUpDown.monitoring.inHomePos;
   "Unit1.Em3.ControlNodes".topTapeAttachment."step".transition1[470] := #_w1 AND "Unit1.Em3.ControlNodes".cmTopTapeAttachmentUpDown.monitoring.inHomePos;
   #statTonTime[470].TON(IN := #_w1 AND "Unit1.Em3.ControlNodes".topTapeAttachment."step".transition1[470],
                         PT := T#100ms);
   IF #statTonTime[470].Q THEN
       "Unit1.Em3.ControlNodes".topTapeAttachment.sequence.status.nextStep := #JOB_4_STEP_80;
   END_IF;
END_REGION

REGION Network 39: Step[480] : Top Tape X-Axis Wait Pos
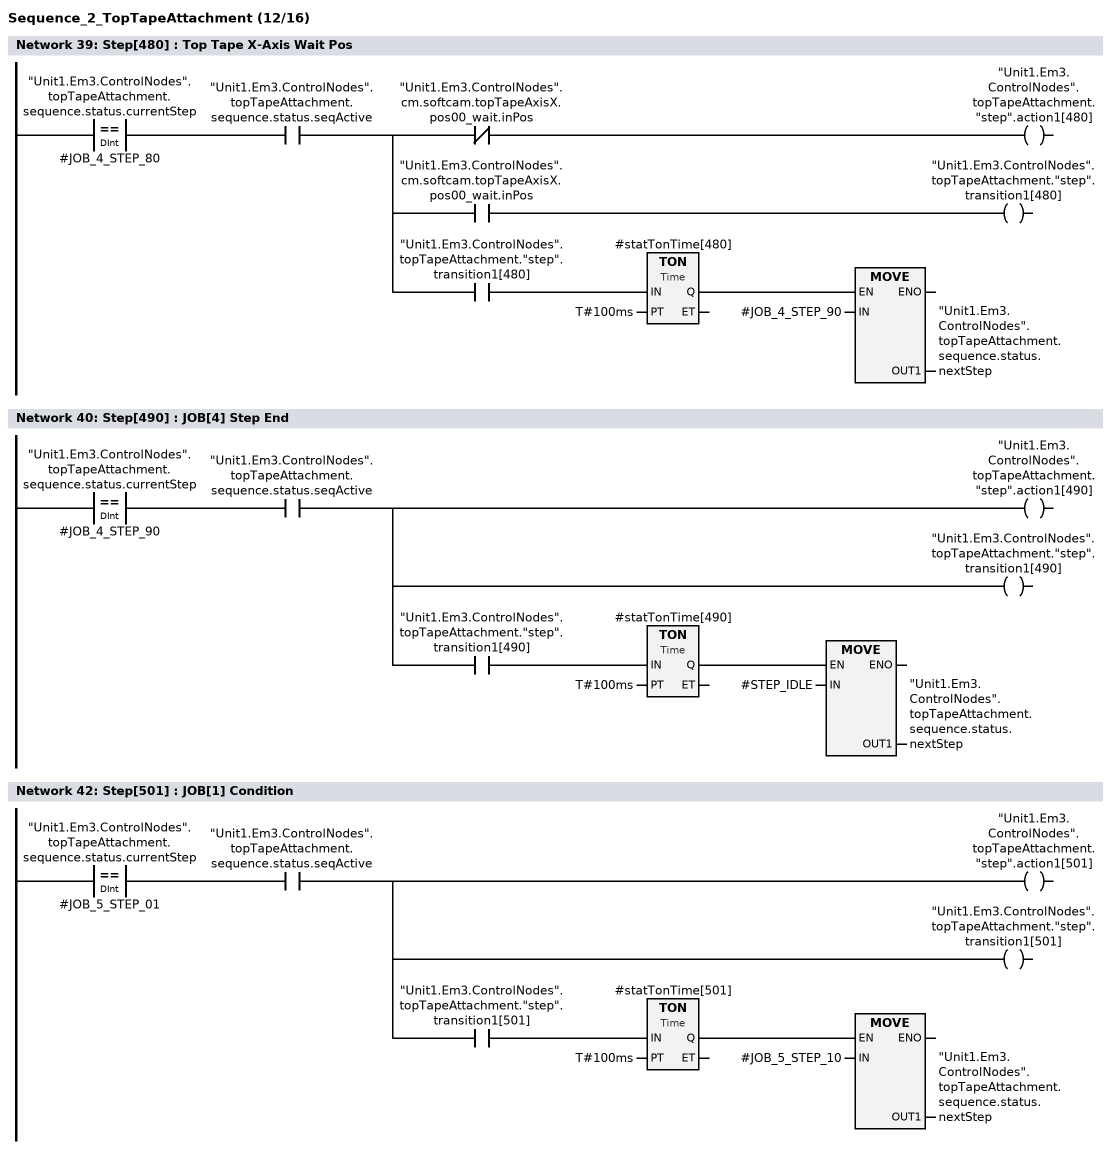
   RUNG wire#powerrail
      { S7_Templates := "SrcType := DInt" } EQ_Contact(in1 := "Unit1.Em3.ControlNodes".topTapeAttachment.sequence.status.currentStep, in2 := #JOB_4_STEP_80)
      Contact( "Unit1.Em3.ControlNodes".topTapeAttachment.sequence.status.seqActive )
      wire#w1
      I_Contact( "Unit1.Em3.ControlNodes".cm.softcam.topTapeAxisX.pos00_wait.inPos )
      Coil( "Unit1.Em3.ControlNodes".topTapeAttachment."step".action1[480] )
   END_RUNG
   RUNG wire#w1
      Contact( "Unit1.Em3.ControlNodes".cm.softcam.topTapeAxisX.pos00_wait.inPos )
      Coil( "Unit1.Em3.ControlNodes".topTapeAttachment."step".transition1[480] )
   END_RUNG
   RUNG wire#w1
      Contact( "Unit1.Em3.ControlNodes".topTapeAttachment."step".transition1[480] )
      { S7_Templates := "time_type := Time" } #statTonTime[480].TON(pt := T#100ms, et =>)
      Move(in := #JOB_4_STEP_90, out1 => "Unit1.Em3.ControlNodes".topTapeAttachment.sequence.status.nextStep)
   END_RUNG
   // the same network as SCL:
   #_w1 := ("Unit1.Em3.ControlNodes".topTapeAttachment.sequence.status.currentStep = #JOB_4_STEP_80) AND "Unit1.Em3.ControlNodes".topTapeAttachment.sequence.status.seqActive;
   "Unit1.Em3.ControlNodes".topTapeAttachment."step".action1[480] := #_w1 AND NOT "Unit1.Em3.ControlNodes".cm.softcam.topTapeAxisX.pos00_wait.inPos;
   "Unit1.Em3.ControlNodes".topTapeAttachment."step".transition1[480] := #_w1 AND "Unit1.Em3.ControlNodes".cm.softcam.topTapeAxisX.pos00_wait.inPos;
   #statTonTime[480].TON(IN := #_w1 AND "Unit1.Em3.ControlNodes".topTapeAttachment."step".transition1[480],
                         PT := T#100ms);
   IF #statTonTime[480].Q THEN
       "Unit1.Em3.ControlNodes".topTapeAttachment.sequence.status.nextStep := #JOB_4_STEP_90;
   END_IF;
END_REGION

REGION Network 40: Step[490] : JOB[4] Step End
   RUNG wire#powerrail
      { S7_Templates := "SrcType := DInt" } EQ_Contact(in1 := "Unit1.Em3.ControlNodes".topTapeAttachment.sequence.status.currentStep, in2 := #JOB_4_STEP_90)
      Contact( "Unit1.Em3.ControlNodes".topTapeAttachment.sequence.status.seqActive )
      wire#w1
      Coil( "Unit1.Em3.ControlNodes".topTapeAttachment."step".action1[490] )
   END_RUNG
   RUNG wire#w1
      Coil( "Unit1.Em3.ControlNodes".topTapeAttachment."step".transition1[490] )
   END_RUNG
   RUNG wire#w1
      Contact( "Unit1.Em3.ControlNodes".topTapeAttachment."step".transition1[490] )
      { S7_Templates := "time_type := Time" } #statTonTime[490].TON(pt := T#100ms, et =>)
      Move(in := #STEP_IDLE, out1 => "Unit1.Em3.ControlNodes".topTapeAttachment.sequence.status.nextStep)
   END_RUNG
   // the same network as SCL:
   "Unit1.Em3.ControlNodes".topTapeAttachment."step".action1[490] := ("Unit1.Em3.ControlNodes".topTapeAttachment.sequence.status.currentStep = #JOB_4_STEP_90) AND "Unit1.Em3.ControlNodes".topTapeAttachment.sequence.status.seqActive;
   "Unit1.Em3.ControlNodes".topTapeAttachment."step".transition1[490] := ("Unit1.Em3.ControlNodes".topTapeAttachment.sequence.status.currentStep = #JOB_4_STEP_90) AND "Unit1.Em3.ControlNodes".topTapeAttachment.sequence.status.seqActive;
   #statTonTime[490].TON(IN := ("Unit1.Em3.ControlNodes".topTapeAttachment.sequence.status.currentStep = #JOB_4_STEP_90) AND "Unit1.Em3.ControlNodes".topTapeAttachment.sequence.status.seqActive AND "Unit1.Em3.ControlNodes".topTapeAttachment."step".transition1[490],
                         PT := T#100ms);
   IF #statTonTime[490].Q THEN
       "Unit1.Em3.ControlNodes".topTapeAttachment.sequence.status.nextStep := #STEP_IDLE;
   END_IF;
END_REGION

REGION Network 41: *************** JOB[5] IDLE STEP_ Throw away tape *************************
END_REGION

REGION Network 42: Step[501] : JOB[1] Condition
   RUNG wire#powerrail
      { S7_Templates := "SrcType := DInt" } EQ_Contact(in1 := "Unit1.Em3.ControlNodes".topTapeAttachment.sequence.status.currentStep, in2 := #JOB_5_STEP_01)
      Contact( "Unit1.Em3.ControlNodes".topTapeAttachment.sequence.status.seqActive )
      wire#w1
      Coil( "Unit1.Em3.ControlNodes".topTapeAttachment."step".action1[501] )
   END_RUNG
   RUNG wire#w1
      Coil( "Unit1.Em3.ControlNodes".topTapeAttachment."step".transition1[501] )
   END_RUNG
   RUNG wire#w1
      Contact( "Unit1.Em3.ControlNodes".topTapeAttachment."step".transition1[501] )
      { S7_Templates := "time_type := Time" } #statTonTime[501].TON(pt := T#100ms, et =>)
      Move(in := #JOB_5_STEP_10, out1 => "Unit1.Em3.ControlNodes".topTapeAttachment.sequence.status.nextStep)
   END_RUNG
   // the same network as SCL:
   "Unit1.Em3.ControlNodes".topTapeAttachment."step".action1[501] := ("Unit1.Em3.ControlNodes".topTapeAttachment.sequence.status.currentStep = #JOB_5_STEP_01) AND "Unit1.Em3.ControlNodes".topTapeAttachment.sequence.status.seqActive;
   "Unit1.Em3.ControlNodes".topTapeAttachment."step".transition1[501] := ("Unit1.Em3.ControlNodes".topTapeAttachment.sequence.status.currentStep = #JOB_5_STEP_01) AND "Unit1.Em3.ControlNodes".topTapeAttachment.sequence.status.seqActive;
   #statTonTime[501].TON(IN := ("Unit1.Em3.ControlNodes".topTapeAttachment.sequence.status.currentStep = #JOB_5_STEP_01) AND "Unit1.Em3.ControlNodes".topTapeAttachment.sequence.status.seqActive AND "Unit1.Em3.ControlNodes".topTapeAttachment."step".transition1[501],
                         PT := T#100ms);
   IF #statTonTime[501].Q THEN
       "Unit1.Em3.ControlNodes".topTapeAttachment.sequence.status.nextStep := #JOB_5_STEP_10;
   END_IF;
END_REGION

REGION Network 43: Step[510] : Attachment Up
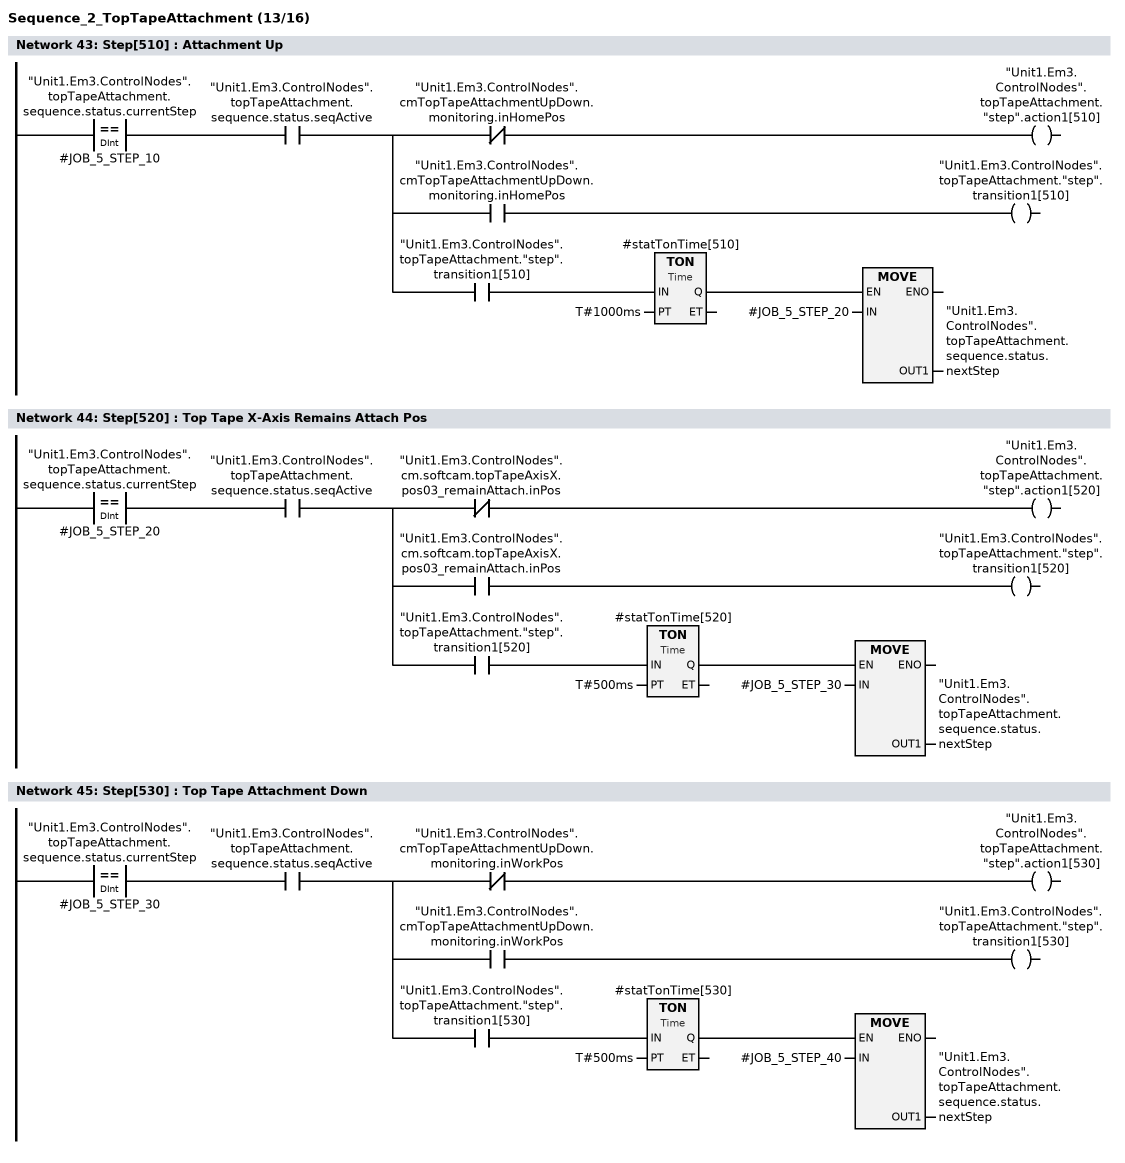
   RUNG wire#powerrail
      { S7_Templates := "SrcType := DInt" } EQ_Contact(in1 := "Unit1.Em3.ControlNodes".topTapeAttachment.sequence.status.currentStep, in2 := #JOB_5_STEP_10)
      Contact( "Unit1.Em3.ControlNodes".topTapeAttachment.sequence.status.seqActive )
      wire#w1
      I_Contact( "Unit1.Em3.ControlNodes".cmTopTapeAttachmentUpDown.monitoring.inHomePos )
      Coil( "Unit1.Em3.ControlNodes".topTapeAttachment."step".action1[510] )
   END_RUNG
   RUNG wire#w1
      Contact( "Unit1.Em3.ControlNodes".cmTopTapeAttachmentUpDown.monitoring.inHomePos )
      Coil( "Unit1.Em3.ControlNodes".topTapeAttachment."step".transition1[510] )
   END_RUNG
   RUNG wire#w1
      Contact( "Unit1.Em3.ControlNodes".topTapeAttachment."step".transition1[510] )
      { S7_Templates := "time_type := Time" } #statTonTime[510].TON(pt := T#1000ms, et =>)
      Move(in := #JOB_5_STEP_20, out1 => "Unit1.Em3.ControlNodes".topTapeAttachment.sequence.status.nextStep)
   END_RUNG
   // the same network as SCL:
   #_w1 := ("Unit1.Em3.ControlNodes".topTapeAttachment.sequence.status.currentStep = #JOB_5_STEP_10) AND "Unit1.Em3.ControlNodes".topTapeAttachment.sequence.status.seqActive;
   "Unit1.Em3.ControlNodes".topTapeAttachment."step".action1[510] := #_w1 AND NOT "Unit1.Em3.ControlNodes".cmTopTapeAttachmentUpDown.monitoring.inHomePos;
   "Unit1.Em3.ControlNodes".topTapeAttachment."step".transition1[510] := #_w1 AND "Unit1.Em3.ControlNodes".cmTopTapeAttachmentUpDown.monitoring.inHomePos;
   #statTonTime[510].TON(IN := #_w1 AND "Unit1.Em3.ControlNodes".topTapeAttachment."step".transition1[510],
                         PT := T#1000ms);
   IF #statTonTime[510].Q THEN
       "Unit1.Em3.ControlNodes".topTapeAttachment.sequence.status.nextStep := #JOB_5_STEP_20;
   END_IF;
END_REGION

REGION Network 44: Step[520] : Top Tape X-Axis Remains Attach Pos
   RUNG wire#powerrail
      { S7_Templates := "SrcType := DInt" } EQ_Contact(in1 := "Unit1.Em3.ControlNodes".topTapeAttachment.sequence.status.currentStep, in2 := #JOB_5_STEP_20)
      Contact( "Unit1.Em3.ControlNodes".topTapeAttachment.sequence.status.seqActive )
      wire#w1
      I_Contact( "Unit1.Em3.ControlNodes".cm.softcam.topTapeAxisX.pos03_remainAttach.inPos )
      Coil( "Unit1.Em3.ControlNodes".topTapeAttachment."step".action1[520] )
   END_RUNG
   RUNG wire#w1
      Contact( "Unit1.Em3.ControlNodes".cm.softcam.topTapeAxisX.pos03_remainAttach.inPos )
      Coil( "Unit1.Em3.ControlNodes".topTapeAttachment."step".transition1[520] )
   END_RUNG
   RUNG wire#w1
      Contact( "Unit1.Em3.ControlNodes".topTapeAttachment."step".transition1[520] )
      { S7_Templates := "time_type := Time" } #statTonTime[520].TON(pt := T#500ms, et =>)
      Move(in := #JOB_5_STEP_30, out1 => "Unit1.Em3.ControlNodes".topTapeAttachment.sequence.status.nextStep)
   END_RUNG
   // the same network as SCL:
   #_w1 := ("Unit1.Em3.ControlNodes".topTapeAttachment.sequence.status.currentStep = #JOB_5_STEP_20) AND "Unit1.Em3.ControlNodes".topTapeAttachment.sequence.status.seqActive;
   "Unit1.Em3.ControlNodes".topTapeAttachment."step".action1[520] := #_w1 AND NOT "Unit1.Em3.ControlNodes".cm.softcam.topTapeAxisX.pos03_remainAttach.inPos;
   "Unit1.Em3.ControlNodes".topTapeAttachment."step".transition1[520] := #_w1 AND "Unit1.Em3.ControlNodes".cm.softcam.topTapeAxisX.pos03_remainAttach.inPos;
   #statTonTime[520].TON(IN := #_w1 AND "Unit1.Em3.ControlNodes".topTapeAttachment."step".transition1[520],
                         PT := T#500ms);
   IF #statTonTime[520].Q THEN
       "Unit1.Em3.ControlNodes".topTapeAttachment.sequence.status.nextStep := #JOB_5_STEP_30;
   END_IF;
END_REGION

REGION Network 45: Step[530] : Top Tape Attachment Down
   RUNG wire#powerrail
      { S7_Templates := "SrcType := DInt" } EQ_Contact(in1 := "Unit1.Em3.ControlNodes".topTapeAttachment.sequence.status.currentStep, in2 := #JOB_5_STEP_30)
      Contact( "Unit1.Em3.ControlNodes".topTapeAttachment.sequence.status.seqActive )
      wire#w1
      I_Contact( "Unit1.Em3.ControlNodes".cmTopTapeAttachmentUpDown.monitoring.inWorkPos )
      Coil( "Unit1.Em3.ControlNodes".topTapeAttachment."step".action1[530] )
   END_RUNG
   RUNG wire#w1
      Contact( "Unit1.Em3.ControlNodes".cmTopTapeAttachmentUpDown.monitoring.inWorkPos )
      Coil( "Unit1.Em3.ControlNodes".topTapeAttachment."step".transition1[530] )
   END_RUNG
   RUNG wire#w1
      Contact( "Unit1.Em3.ControlNodes".topTapeAttachment."step".transition1[530] )
      { S7_Templates := "time_type := Time" } #statTonTime[530].TON(pt := T#500ms, et =>)
      Move(in := #JOB_5_STEP_40, out1 => "Unit1.Em3.ControlNodes".topTapeAttachment.sequence.status.nextStep)
   END_RUNG
   // the same network as SCL:
   #_w1 := ("Unit1.Em3.ControlNodes".topTapeAttachment.sequence.status.currentStep = #JOB_5_STEP_30) AND "Unit1.Em3.ControlNodes".topTapeAttachment.sequence.status.seqActive;
   "Unit1.Em3.ControlNodes".topTapeAttachment."step".action1[530] := #_w1 AND NOT "Unit1.Em3.ControlNodes".cmTopTapeAttachmentUpDown.monitoring.inWorkPos;
   "Unit1.Em3.ControlNodes".topTapeAttachment."step".transition1[530] := #_w1 AND "Unit1.Em3.ControlNodes".cmTopTapeAttachmentUpDown.monitoring.inWorkPos;
   #statTonTime[530].TON(IN := #_w1 AND "Unit1.Em3.ControlNodes".topTapeAttachment."step".transition1[530],
                         PT := T#500ms);
   IF #statTonTime[530].Q THEN
       "Unit1.Em3.ControlNodes".topTapeAttachment.sequence.status.nextStep := #JOB_5_STEP_40;
   END_IF;
END_REGION

REGION Network 46: Step[540] : Top Tape Attachment Vaccum Off
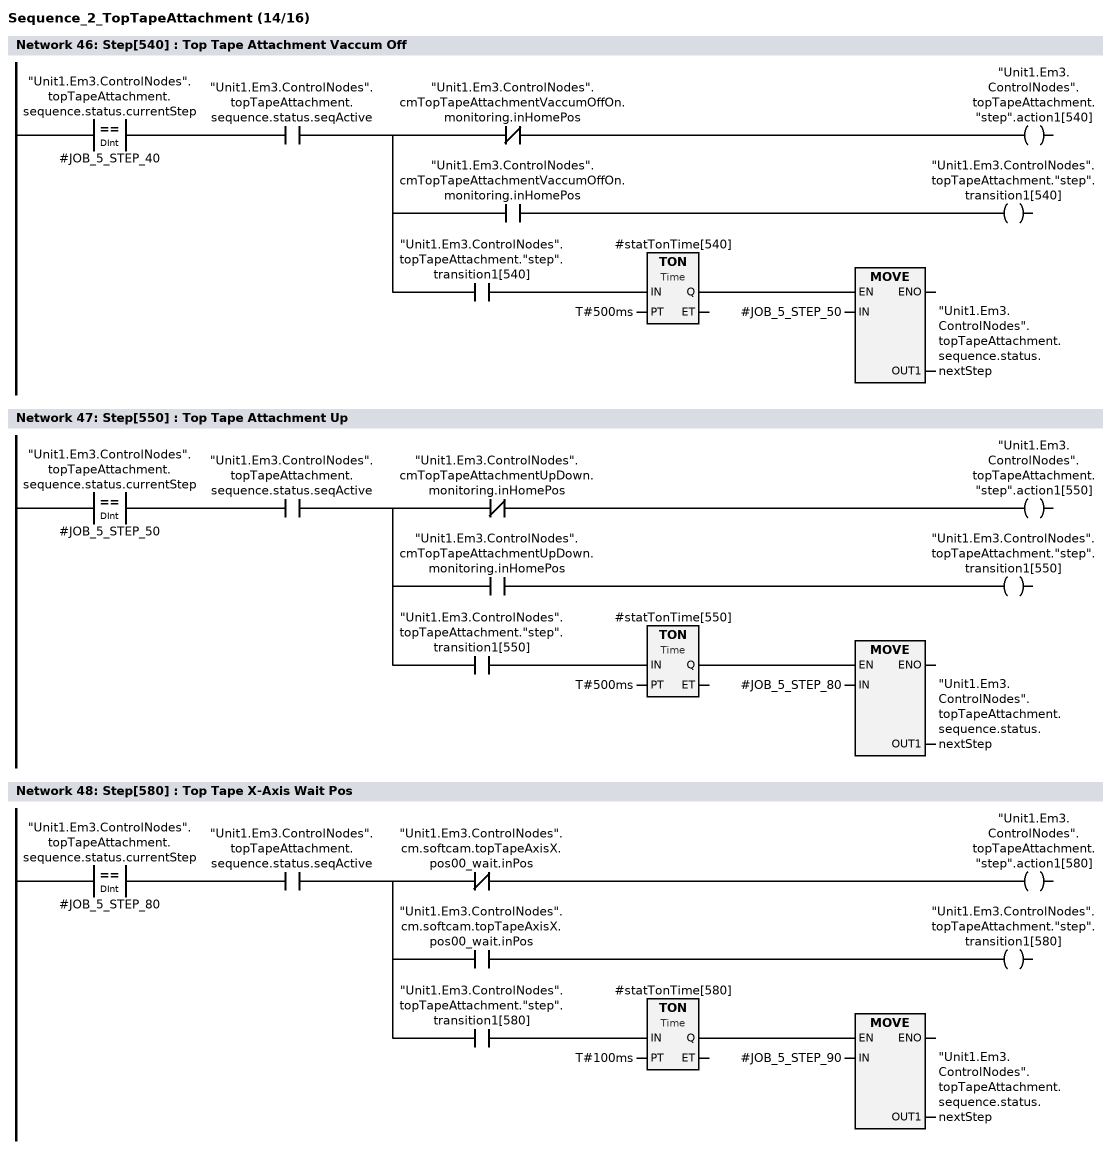
   RUNG wire#powerrail
      { S7_Templates := "SrcType := DInt" } EQ_Contact(in1 := "Unit1.Em3.ControlNodes".topTapeAttachment.sequence.status.currentStep, in2 := #JOB_5_STEP_40)
      Contact( "Unit1.Em3.ControlNodes".topTapeAttachment.sequence.status.seqActive )
      wire#w1
      I_Contact( "Unit1.Em3.ControlNodes".cmTopTapeAttachmentVaccumOffOn.monitoring.inHomePos )
      Coil( "Unit1.Em3.ControlNodes".topTapeAttachment."step".action1[540] )
   END_RUNG
   RUNG wire#w1
      Contact( "Unit1.Em3.ControlNodes".cmTopTapeAttachmentVaccumOffOn.monitoring.inHomePos )
      Coil( "Unit1.Em3.ControlNodes".topTapeAttachment."step".transition1[540] )
   END_RUNG
   RUNG wire#w1
      Contact( "Unit1.Em3.ControlNodes".topTapeAttachment."step".transition1[540] )
      { S7_Templates := "time_type := Time" } #statTonTime[540].TON(pt := T#500ms, et =>)
      Move(in := #JOB_5_STEP_50, out1 => "Unit1.Em3.ControlNodes".topTapeAttachment.sequence.status.nextStep)
   END_RUNG
   // the same network as SCL:
   #_w1 := ("Unit1.Em3.ControlNodes".topTapeAttachment.sequence.status.currentStep = #JOB_5_STEP_40) AND "Unit1.Em3.ControlNodes".topTapeAttachment.sequence.status.seqActive;
   "Unit1.Em3.ControlNodes".topTapeAttachment."step".action1[540] := #_w1 AND NOT "Unit1.Em3.ControlNodes".cmTopTapeAttachmentVaccumOffOn.monitoring.inHomePos;
   "Unit1.Em3.ControlNodes".topTapeAttachment."step".transition1[540] := #_w1 AND "Unit1.Em3.ControlNodes".cmTopTapeAttachmentVaccumOffOn.monitoring.inHomePos;
   #statTonTime[540].TON(IN := #_w1 AND "Unit1.Em3.ControlNodes".topTapeAttachment."step".transition1[540],
                         PT := T#500ms);
   IF #statTonTime[540].Q THEN
       "Unit1.Em3.ControlNodes".topTapeAttachment.sequence.status.nextStep := #JOB_5_STEP_50;
   END_IF;
END_REGION

REGION Network 47: Step[550] : Top Tape Attachment Up
   RUNG wire#powerrail
      { S7_Templates := "SrcType := DInt" } EQ_Contact(in1 := "Unit1.Em3.ControlNodes".topTapeAttachment.sequence.status.currentStep, in2 := #JOB_5_STEP_50)
      Contact( "Unit1.Em3.ControlNodes".topTapeAttachment.sequence.status.seqActive )
      wire#w1
      I_Contact( "Unit1.Em3.ControlNodes".cmTopTapeAttachmentUpDown.monitoring.inHomePos )
      Coil( "Unit1.Em3.ControlNodes".topTapeAttachment."step".action1[550] )
   END_RUNG
   RUNG wire#w1
      Contact( "Unit1.Em3.ControlNodes".cmTopTapeAttachmentUpDown.monitoring.inHomePos )
      Coil( "Unit1.Em3.ControlNodes".topTapeAttachment."step".transition1[550] )
   END_RUNG
   RUNG wire#w1
      Contact( "Unit1.Em3.ControlNodes".topTapeAttachment."step".transition1[550] )
      { S7_Templates := "time_type := Time" } #statTonTime[550].TON(pt := T#500ms, et =>)
      Move(in := #JOB_5_STEP_80, out1 => "Unit1.Em3.ControlNodes".topTapeAttachment.sequence.status.nextStep)
   END_RUNG
   // the same network as SCL:
   #_w1 := ("Unit1.Em3.ControlNodes".topTapeAttachment.sequence.status.currentStep = #JOB_5_STEP_50) AND "Unit1.Em3.ControlNodes".topTapeAttachment.sequence.status.seqActive;
   "Unit1.Em3.ControlNodes".topTapeAttachment."step".action1[550] := #_w1 AND NOT "Unit1.Em3.ControlNodes".cmTopTapeAttachmentUpDown.monitoring.inHomePos;
   "Unit1.Em3.ControlNodes".topTapeAttachment."step".transition1[550] := #_w1 AND "Unit1.Em3.ControlNodes".cmTopTapeAttachmentUpDown.monitoring.inHomePos;
   #statTonTime[550].TON(IN := #_w1 AND "Unit1.Em3.ControlNodes".topTapeAttachment."step".transition1[550],
                         PT := T#500ms);
   IF #statTonTime[550].Q THEN
       "Unit1.Em3.ControlNodes".topTapeAttachment.sequence.status.nextStep := #JOB_5_STEP_80;
   END_IF;
END_REGION

REGION Network 48: Step[580] : Top Tape X-Axis Wait Pos
   RUNG wire#powerrail
      { S7_Templates := "SrcType := DInt" } EQ_Contact(in1 := "Unit1.Em3.ControlNodes".topTapeAttachment.sequence.status.currentStep, in2 := #JOB_5_STEP_80)
      Contact( "Unit1.Em3.ControlNodes".topTapeAttachment.sequence.status.seqActive )
      wire#w1
      I_Contact( "Unit1.Em3.ControlNodes".cm.softcam.topTapeAxisX.pos00_wait.inPos )
      Coil( "Unit1.Em3.ControlNodes".topTapeAttachment."step".action1[580] )
   END_RUNG
   RUNG wire#w1
      Contact( "Unit1.Em3.ControlNodes".cm.softcam.topTapeAxisX.pos00_wait.inPos )
      Coil( "Unit1.Em3.ControlNodes".topTapeAttachment."step".transition1[580] )
   END_RUNG
   RUNG wire#w1
      Contact( "Unit1.Em3.ControlNodes".topTapeAttachment."step".transition1[580] )
      { S7_Templates := "time_type := Time" } #statTonTime[580].TON(pt := T#100ms, et =>)
      Move(in := #JOB_5_STEP_90, out1 => "Unit1.Em3.ControlNodes".topTapeAttachment.sequence.status.nextStep)
   END_RUNG
   // the same network as SCL:
   #_w1 := ("Unit1.Em3.ControlNodes".topTapeAttachment.sequence.status.currentStep = #JOB_5_STEP_80) AND "Unit1.Em3.ControlNodes".topTapeAttachment.sequence.status.seqActive;
   "Unit1.Em3.ControlNodes".topTapeAttachment."step".action1[580] := #_w1 AND NOT "Unit1.Em3.ControlNodes".cm.softcam.topTapeAxisX.pos00_wait.inPos;
   "Unit1.Em3.ControlNodes".topTapeAttachment."step".transition1[580] := #_w1 AND "Unit1.Em3.ControlNodes".cm.softcam.topTapeAxisX.pos00_wait.inPos;
   #statTonTime[580].TON(IN := #_w1 AND "Unit1.Em3.ControlNodes".topTapeAttachment."step".transition1[580],
                         PT := T#100ms);
   IF #statTonTime[580].Q THEN
       "Unit1.Em3.ControlNodes".topTapeAttachment.sequence.status.nextStep := #JOB_5_STEP_90;
   END_IF;
END_REGION

REGION Network 49: Step[590] : JOB[5] Step End
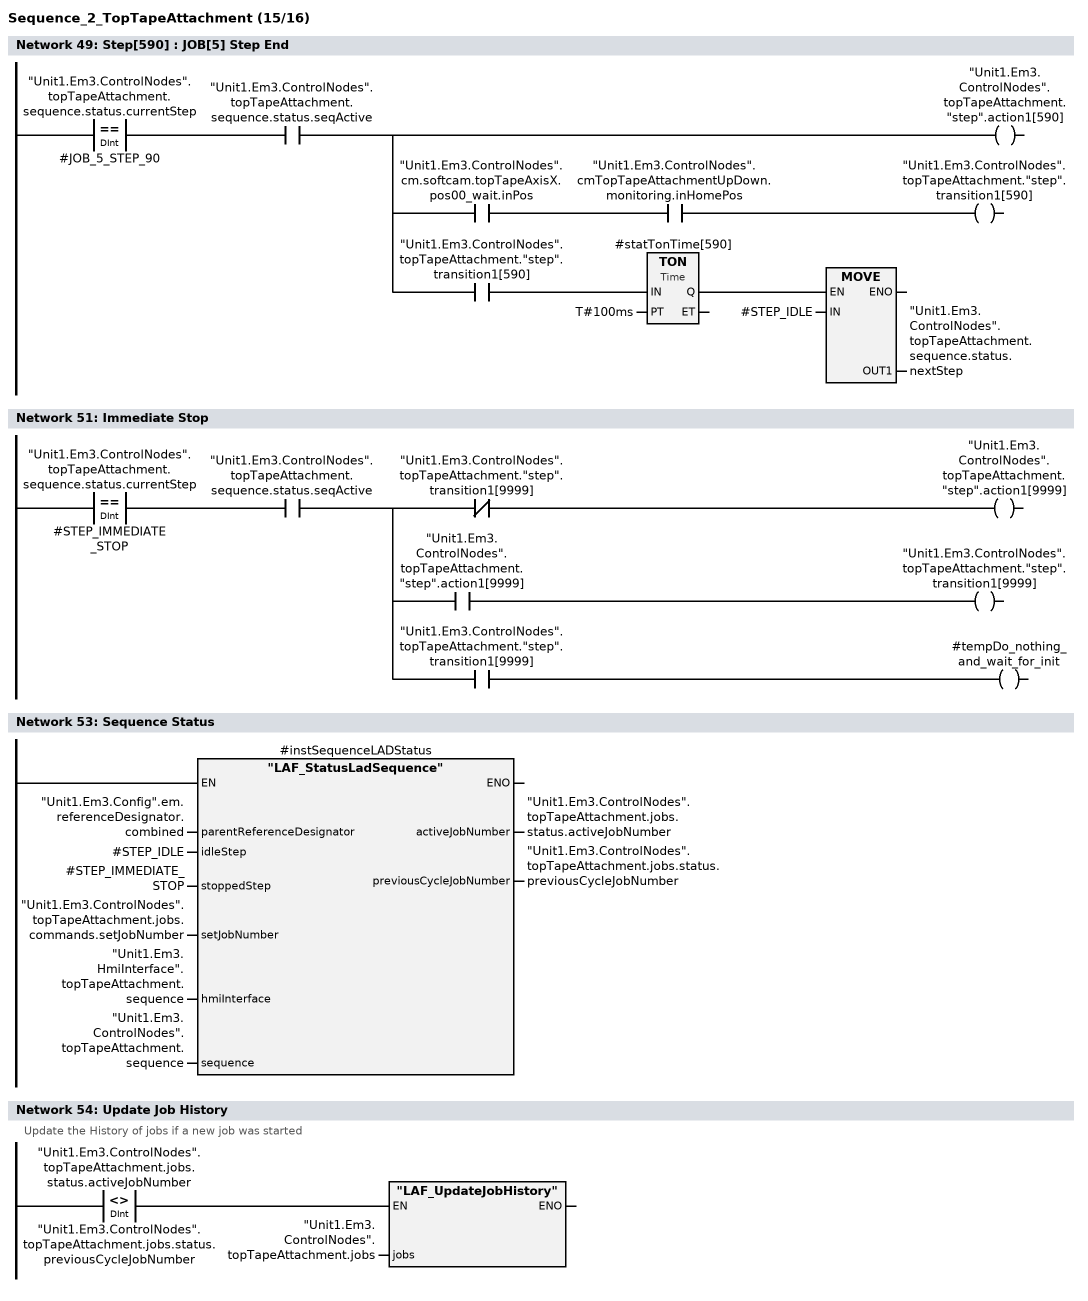
   RUNG wire#powerrail
      { S7_Templates := "SrcType := DInt" } EQ_Contact(in1 := "Unit1.Em3.ControlNodes".topTapeAttachment.sequence.status.currentStep, in2 := #JOB_5_STEP_90)
      Contact( "Unit1.Em3.ControlNodes".topTapeAttachment.sequence.status.seqActive )
      wire#w1
      Coil( "Unit1.Em3.ControlNodes".topTapeAttachment."step".action1[590] )
   END_RUNG
   RUNG wire#w1
      Contact( "Unit1.Em3.ControlNodes".cm.softcam.topTapeAxisX.pos00_wait.inPos )
      Contact( "Unit1.Em3.ControlNodes".cmTopTapeAttachmentUpDown.monitoring.inHomePos )
      Coil( "Unit1.Em3.ControlNodes".topTapeAttachment."step".transition1[590] )
   END_RUNG
   RUNG wire#w1
      Contact( "Unit1.Em3.ControlNodes".topTapeAttachment."step".transition1[590] )
      { S7_Templates := "time_type := Time" } #statTonTime[590].TON(pt := T#100ms, et =>)
      Move(in := #STEP_IDLE, out1 => "Unit1.Em3.ControlNodes".topTapeAttachment.sequence.status.nextStep)
   END_RUNG
   // the same network as SCL:
   "Unit1.Em3.ControlNodes".topTapeAttachment."step".action1[590] := ("Unit1.Em3.ControlNodes".topTapeAttachment.sequence.status.currentStep = #JOB_5_STEP_90) AND "Unit1.Em3.ControlNodes".topTapeAttachment.sequence.status.seqActive;
   "Unit1.Em3.ControlNodes".topTapeAttachment."step".transition1[590] := ("Unit1.Em3.ControlNodes".topTapeAttachment.sequence.status.currentStep = #JOB_5_STEP_90) AND "Unit1.Em3.ControlNodes".topTapeAttachment.sequence.status.seqActive AND "Unit1.Em3.ControlNodes".cm.softcam.topTapeAxisX.pos00_wait.inPos AND "Unit1.Em3.ControlNodes".cmTopTapeAttachmentUpDown.monitoring.inHomePos;
   #statTonTime[590].TON(IN := ("Unit1.Em3.ControlNodes".topTapeAttachment.sequence.status.currentStep = #JOB_5_STEP_90) AND "Unit1.Em3.ControlNodes".topTapeAttachment.sequence.status.seqActive AND "Unit1.Em3.ControlNodes".topTapeAttachment."step".transition1[590],
                         PT := T#100ms);
   IF #statTonTime[590].Q THEN
       "Unit1.Em3.ControlNodes".topTapeAttachment.sequence.status.nextStep := #STEP_IDLE;
   END_IF;
END_REGION

REGION Network 50: *************** IMMEDIATE STOP ****************
END_REGION

REGION Network 51: Immediate Stop
   RUNG wire#powerrail
      { S7_Templates := "SrcType := DInt" } EQ_Contact(in1 := "Unit1.Em3.ControlNodes".topTapeAttachment.sequence.status.currentStep, in2 := #STEP_IMMEDIATE_STOP)
      Contact( "Unit1.Em3.ControlNodes".topTapeAttachment.sequence.status.seqActive )
      wire#w1
      I_Contact( "Unit1.Em3.ControlNodes".topTapeAttachment."step".transition1[9999] )
      Coil( "Unit1.Em3.ControlNodes".topTapeAttachment."step".action1[9999] )
   END_RUNG
   RUNG wire#w1
      Contact( "Unit1.Em3.ControlNodes".topTapeAttachment."step".action1[9999] )
      Coil( "Unit1.Em3.ControlNodes".topTapeAttachment."step".transition1[9999] )
   END_RUNG
   RUNG wire#w1
      Contact( "Unit1.Em3.ControlNodes".topTapeAttachment."step".transition1[9999] )
      Coil( #tempDo_nothing_and_wait_for_init )
   END_RUNG
   // the same network as SCL:
   #_w1 := ("Unit1.Em3.ControlNodes".topTapeAttachment.sequence.status.currentStep = #STEP_IMMEDIATE_STOP) AND "Unit1.Em3.ControlNodes".topTapeAttachment.sequence.status.seqActive;
   "Unit1.Em3.ControlNodes".topTapeAttachment."step".action1[9999] := #_w1 AND NOT "Unit1.Em3.ControlNodes".topTapeAttachment."step".transition1[9999];
   "Unit1.Em3.ControlNodes".topTapeAttachment."step".transition1[9999] := #_w1 AND "Unit1.Em3.ControlNodes".topTapeAttachment."step".action1[9999];
   #tempDo_nothing_and_wait_for_init := #_w1 AND "Unit1.Em3.ControlNodes".topTapeAttachment."step".transition1[9999];
END_REGION

REGION Network 52: *************** STATUS **********************
END_REGION

REGION Network 53: Sequence Status
   RUNG wire#powerrail
      #instSequenceLADStatus(parentReferenceDesignator := "Unit1.Em3.Config".em.referenceDesignator.combined, idleStep := #STEP_IDLE, stoppedStep := #STEP_IMMEDIATE_STOP, setJobNumber := "Unit1.Em3.ControlNodes".topTapeAttachment.jobs.commands.setJobNumber, hmiInterface := "Unit1.Em3.HmiInterface".topTapeAttachment.sequence, sequence := "Unit1.Em3.ControlNodes".topTapeAttachment.sequence, activeJobNumber => "Unit1.Em3.ControlNodes".topTapeAttachment.jobs.status.activeJobNumber, previousCycleJobNumber => "Unit1.Em3.ControlNodes".topTapeAttachment.jobs.status.previousCycleJobNumber)
   END_RUNG
   // the same network as SCL:
   #instSequenceLADStatus(parentReferenceDesignator := "Unit1.Em3.Config".em.referenceDesignator.combined,   // "LAF_StatusLadSequence"
                          idleStep := #STEP_IDLE,
                          stoppedStep := #STEP_IMMEDIATE_STOP,
                          setJobNumber := "Unit1.Em3.ControlNodes".topTapeAttachment.jobs.commands.setJobNumber,
                          hmiInterface := "Unit1.Em3.HmiInterface".topTapeAttachment.sequence,
                          sequence := "Unit1.Em3.ControlNodes".topTapeAttachment.sequence,
                          activeJobNumber => "Unit1.Em3.ControlNodes".topTapeAttachment.jobs.status.activeJobNumber,
                          previousCycleJobNumber => "Unit1.Em3.ControlNodes".topTapeAttachment.jobs.status.previousCycleJobNumber);
END_REGION

REGION Network 54: Update Job History
   // Update the History of jobs if a new job was started
   RUNG wire#powerrail
      { S7_Templates := "SrcType := DInt" } NE_Contact(in1 := "Unit1.Em3.ControlNodes".topTapeAttachment.jobs.status.activeJobNumber, in2 := "Unit1.Em3.ControlNodes".topTapeAttachment.jobs.status.previousCycleJobNumber)
      "LAF_UpdateJobHistory"(jobs := "Unit1.Em3.ControlNodes".topTapeAttachment.jobs)
   END_RUNG
   // the same network as SCL:
   IF "Unit1.Em3.ControlNodes".topTapeAttachment.jobs.status.activeJobNumber <> "Unit1.Em3.ControlNodes".topTapeAttachment.jobs.status.previousCycleJobNumber THEN
       "LAF_UpdateJobHistory"(jobs := "Unit1.Em3.ControlNodes".topTapeAttachment.jobs);
   END_IF;
END_REGION

REGION Network 55: Output steps as String
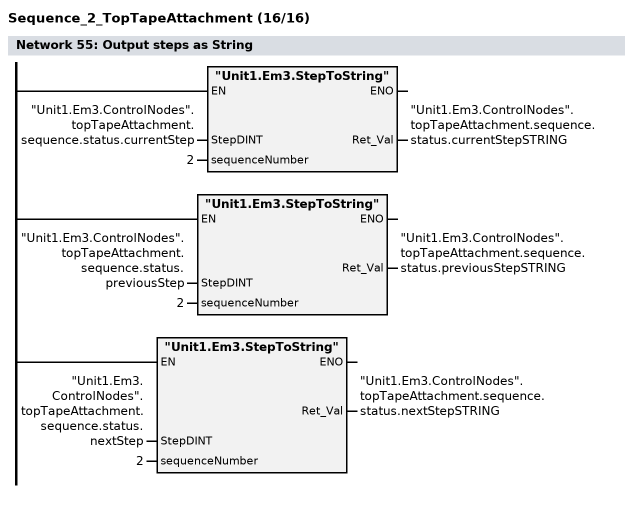
   RUNG wire#powerrail
      "Unit1.Em3.StepToString"(StepDINT := "Unit1.Em3.ControlNodes".topTapeAttachment.sequence.status.currentStep, sequenceNumber := 2, Ret_Val => "Unit1.Em3.ControlNodes".topTapeAttachment.sequence.status.currentStepSTRING)
   END_RUNG
   RUNG wire#powerrail
      "Unit1.Em3.StepToString"(StepDINT := "Unit1.Em3.ControlNodes".topTapeAttachment.sequence.status.previousStep, sequenceNumber := 2, Ret_Val => "Unit1.Em3.ControlNodes".topTapeAttachment.sequence.status.previousStepSTRING)
   END_RUNG
   RUNG wire#powerrail
      "Unit1.Em3.StepToString"(StepDINT := "Unit1.Em3.ControlNodes".topTapeAttachment.sequence.status.nextStep, sequenceNumber := 2, Ret_Val => "Unit1.Em3.ControlNodes".topTapeAttachment.sequence.status.nextStepSTRING)
   END_RUNG
   // the same network as SCL:
   "Unit1.Em3.ControlNodes".topTapeAttachment.sequence.status.currentStepSTRING := "Unit1.Em3.StepToString"(StepDINT := "Unit1.Em3.ControlNodes".topTapeAttachment.sequence.status.currentStep,
                           sequenceNumber := 2);
   "Unit1.Em3.ControlNodes".topTapeAttachment.sequence.status.previousStepSTRING := "Unit1.Em3.StepToString"(StepDINT := "Unit1.Em3.ControlNodes".topTapeAttachment.sequence.status.previousStep,
                           sequenceNumber := 2);
   "Unit1.Em3.ControlNodes".topTapeAttachment.sequence.status.nextStepSTRING := "Unit1.Em3.StepToString"(StepDINT := "Unit1.Em3.ControlNodes".topTapeAttachment.sequence.status.nextStep,
                           sequenceNumber := 2);
END_REGION
END_FUNCTION_BLOCK
